LIN {X 0,Y 656.693,Z 410.418,A -85,B 0,C 180,E1 30799.109,E2 30799.109} C_VEL
LIN {X 0,Y 656.695,Z 410.425,A -85,B 0,C 180,E1 30796.088,E2 30796.088} C_VEL
LIN {X 0,Y 656.69,Z 410.427,A -85,B 0,C 180,E1 30793.023,E2 30793.023} C_VEL
LIN {X 0,Y 656.7,Z 410.423,A -85,B 0,C 180,E1 30789.996,E2 30789.996} C_VEL
LIN {X 0,Y 656.683,Z 410.43,A -85,B 0,C 180,E1 30786.896,E2 30786.896} C_VEL
LIN {X 0,Y 656.702,Z 410.42,A -85,B 0,C 180,E1 30783.841,E2 30783.841} C_VEL
LIN {X 0,Y 656.676,Z 410.43,A -85,B 0,C 180,E1 30780.785,E2 30780.785} C_VEL
LIN {X 0,Y 656.705,Z 410.416,A -85,B 0,C 180,E1 30777.819,E2 30777.819} C_VEL
LIN {X 0,Y 656.671,Z 410.43,A -85,B 0,C 180,E1 30774.758,E2 30774.758} C_VEL
LIN {X 0,Y 656.707,Z 410.411,A -85,B 0,C 180,E1 30771.763,E2 30771.763} C_VEL
LIN {X 0,Y 656.665,Z 410.429,A -85,B 0,C 180,E1 30768.672,E2 30768.672} C_VEL
LIN {X 0,Y 656.702,Z 410.411,A -85,B 0,C 180,E1 30765.72,E2 30765.72} C_VEL
LIN {X 0,Y 656.661,Z 410.426,A -85,B 0,C 180,E1 30762.636,E2 30762.636} C_VEL
LIN {X 0,Y 656.679,Z 410.421,A -85,B 0,C 180,E1 30759.779,E2 30759.779} C_VEL
LIN {X 0,Y 656.66,Z 410.417,A -85,B 0,C 180,E1 30756.663,E2 30756.663} C_VEL
LIN {X 0,Y 656.653,Z 410.429,A -85,B 0,C 180,E1 30753.892,E2 30753.892} C_VEL
LIN {X 0,Y 656.668,Z 410.427,A -85,B 0,C 180,E1 30750.74,E2 30750.74} C_VEL
LIN {X 0,Y 656.635,Z 410.428,A -85,B 0,C 180,E1 30748,E2 30748} C_VEL
LIN {X 0,Y 656.698,Z 410.433,A -85,B 0,C 180,E1 30744.969,E2 30744.969} C_VEL
LIN {X 0,Y 656.625,Z 410.434,A -85,B 0,C 180,E1 30742.074,E2 30742.074} C_VEL
LIN {X 0,Y 656.649,Z 410.429,A -85,B 0,C 180,E1 30740.539,E2 30740.539} C_VEL
LIN {X 0,Y 655.6,Z 410.557,A -85,B 0,C 180,E1 30739.867,E2 30739.867} C_VEL
LIN {X 0,Y 649.187,Z 411.313,A -85,B 0,C 180,E1 30737.983,E2 30737.983} C_VEL
LIN {X 0,Y 648.697,Z 411.374,A -85,B 0,C 180,E1 30737.493,E2 30737.493} C_VEL
LIN {X 0,Y 648.686,Z 411.423,A -85,B 0,C 180,E1 30734.288,E2 30734.288} C_VEL
LIN {X 0,Y 648.673,Z 411.379,A -85,B 0,C 180,E1 30731.617,E2 30731.617} C_VEL
LIN {X 0,Y 648.721,Z 411.408,A -85,B 0,C 180,E1 30728.606,E2 30728.606} C_VEL
LIN {X 0,Y 648.773,Z 411.633,A -85,B 0,C 180,E1 30726.726,E2 30726.726} C_VEL
LIN {X 0,Y 650.211,Z 415.779,A -85,B 0,C 180,E1 30726.237,E2 30726.237} C_VEL
LIN {X 0,Y 662.995,Z 436.741,A -85,B 0,C 180,E1 30725.041,E2 30725.041} C_VEL
LIN {X 0,Y 667.932,Z 445.525,A -85,B 0,C 180,E1 30724.59,E2 30724.59} C_VEL
LIN {X 0,Y 664.816,Z 693.939,A -85,B 0,C 180,E1 30721.53,E2 30721.53} C_VEL
LIN {X 0,Y 663.436,Z 804.05,A -85,B 0,C 180,E1 30720.173,E2 30720.173} C_VEL
LIN {X 0,Y 662.695,Z 829.21,A -85,B 0,C 180,E1 30719.71,E2 30719.71} C_VEL
LIN {X 0,Y 661.876,Z 849.807,A -85,B 0,C 180,E1 30719.2,E2 30719.2} C_VEL
LIN {X 0,Y 660.879,Z 872.181,A -85,B 0,C 180,E1 30718.512,E2 30718.512} C_VEL
LIN {X 0,Y 659.671,Z 893.971,A -85,B 0,C 180,E1 30717.683,E2 30717.683} C_VEL
LIN {X 0,Y 658.517,Z 914.637,A -85,B 0,C 180,E1 30716.757,E2 30716.757} C_VEL
LIN {X 0,Y 657.055,Z 937.416,A -85,B 0,C 180,E1 30715.553,E2 30715.553} C_VEL
LIN {X 0,Y 655.807,Z 956.221,A -85,B 0,C 180,E1 30714.405,E2 30714.405} C_VEL
LIN {X 0,Y 654.415,Z 977.19,A -85,B 0,C 180,E1 30712.931,E2 30712.931} C_VEL
LIN {X 0,Y 653.234,Z 994.357,A -85,B 0,C 180,E1 30711.553,E2 30711.553} C_VEL
LIN {X 0,Y 652.004,Z 1013.415,A -85,B 0,C 180,E1 30709.811,E2 30709.811} C_VEL
LIN {X 0,Y 651.067,Z 1028.308,A -85,B 0,C 180,E1 30708.258,E2 30708.258} C_VEL
LIN {X 0,Y 650.158,Z 1044.481,A -85,B 0,C 180,E1 30706.346,E2 30706.346} C_VEL
LIN {X 0,Y 649.48,Z 1057.15,A -85,B 0,C 180,E1 30704.625,E2 30704.625} C_VEL
LIN {X 0,Y 648.926,Z 1069.98,A -85,B 0,C 180,E1 30702.639,E2 30702.639} C_VEL
LIN {X 0,Y 648.524,Z 1080.788,A -85,B 0,C 180,E1 30700.662,E2 30700.662} C_VEL
LIN {X 0,Y 648.247,Z 1090.431,A -85,B 0,C 180,E1 30698.605,E2 30698.605} C_VEL
LIN {X 0,Y 648.052,Z 1098.176,A -85,B 0,C 180,E1 30696.556,E2 30696.556} C_VEL
LIN {X 0,Y 647.96,Z 1103.94,A -85,B 0,C 180,E1 30694.691,E2 30694.691} C_VEL
LIN {X 0,Y 647.925,Z 1109.279,A -85,B 0,C 180,E1 30692.388,E2 30692.388} C_VEL
LIN {X 0,Y 647.914,Z 1112.302,A -85,B 0,C 180,E1 30690.442,E2 30690.442} C_VEL
LIN {X 0,Y 647.894,Z 1114.159,A -85,B 0,C 180,E1 30688.32,E2 30688.32} C_VEL
LIN {X 0,Y 647.892,Z 1114.337,A -85,B 0,C 180,E1 30686.284,E2 30686.284} C_VEL
LIN {X 0,Y 647.905,Z 1113.249,A -85,B 0,C 180,E1 30684.332,E2 30684.332} C_VEL
LIN {X 0,Y 647.924,Z 1110.328,A -85,B 0,C 180,E1 30682.106,E2 30682.106} C_VEL
LIN {X 0,Y 647.93,Z 1106.499,A -85,B 0,C 180,E1 30680.227,E2 30680.227} C_VEL
LIN {X 0,Y 647.996,Z 1100.901,A -85,B 0,C 180,E1 30678.157,E2 30678.157} C_VEL
LIN {X 0,Y 648.149,Z 1093.476,A -85,B 0,C 180,E1 30676.074,E2 30676.074} C_VEL
LIN {X 0,Y 648.371,Z 1085.278,A -85,B 0,C 180,E1 30674.159,E2 30674.159} C_VEL
LIN {X 0,Y 648.734,Z 1074.384,A -85,B 0,C 180,E1 30672.046,E2 30672.046} C_VEL
LIN {X 0,Y 649.186,Z 1063.508,A -85,B 0,C 180,E1 30670.234,E2 30670.234} C_VEL
LIN {X 0,Y 649.864,Z 1049.605,A -85,B 0,C 180,E1 30668.235,E2 30668.235} C_VEL
LIN {X 0,Y 650.618,Z 1036.132,A -85,B 0,C 180,E1 30666.544,E2 30666.544} C_VEL
LIN {X 0,Y 651.643,Z 1018.935,A -85,B 0,C 180,E1 30664.653,E2 30664.653} C_VEL
LIN {X 0,Y 652.668,Z 1003.148,A -85,B 0,C 180,E1 30663.132,E2 30663.132} C_VEL
LIN {X 0,Y 653.958,Z 983.638,A -85,B 0,C 180,E1 30661.474,E2 30661.474} C_VEL
LIN {X 0,Y 655.214,Z 965.251,A -85,B 0,C 180,E1 30660.115,E2 30660.115} C_VEL
LIN {X 0,Y 656.661,Z 943.663,A -85,B 0,C 180,E1 30658.719,E2 30658.719} C_VEL
LIN {X 0,Y 657.924,Z 923.66,A -85,B 0,C 180,E1 30657.607,E2 30657.607} C_VEL
LIN {X 0,Y 659.328,Z 900.994,A -85,B 0,C 180,E1 30656.522,E2 30656.522} C_VEL
LIN {X 0,Y 660.467,Z 879.681,A -85,B 0,C 180,E1 30655.672,E2 30655.672} C_VEL
LIN {X 0,Y 661.604,Z 856.553,A -85,B 0,C 180,E1 30654.896,E2 30654.896} C_VEL
LIN {X 0,Y 662.536,Z 832.984,A -85,B 0,C 180,E1 30654.285,E2 30654.285} C_VEL
LIN {X 0,Y 663.294,Z 810.621,A -85,B 0,C 180,E1 30653.841,E2 30653.841} C_VEL
LIN {X 0,Y 663.84,Z 776.914,A -85,B 0,C 180,E1 30653.386,E2 30653.386} C_VEL
LIN {X 0,Y 666.852,Z 528.949,A -85,B 0,C 180,E1 30650.355,E2 30650.355} C_VEL
LIN {X 0,Y 667.836,Z 445.069,A -85,B 0,C 180,E1 30649.307,E2 30649.307} C_VEL
LIN {X 0,Y 654.643,Z 422.915,A -85,B 0,C 180,E1 30648.092,E2 30648.092} C_VEL
LIN {X 0,Y 650.084,Z 415.41,A -85,B 0,C 180,E1 30647.628,E2 30647.628} C_VEL
LIN {X 0,Y 648.768,Z 411.552,A -85,B 0,C 180,E1 30647.121,E2 30647.121} C_VEL
LIN {X 0,Y 648.675,Z 411.43,A -85,B 0,C 180,E1 30644.165,E2 30644.165} C_VEL
LIN {X 0,Y 648.698,Z 411.385,A -85,B 0,C 180,E1 30641.486,E2 30641.486} C_VEL
LIN {X 0,Y 648.696,Z 411.42,A -85,B 0,C 180,E1 30638.319,E2 30638.319} C_VEL
LIN {X 0,Y 648.687,Z 411.38,A -85,B 0,C 180,E1 30635.637,E2 30635.637} C_VEL
LIN {X 0,Y 648.737,Z 411.417,A -85,B 0,C 180,E1 30632.532,E2 30632.532} C_VEL
LIN {X 0,Y 648.69,Z 411.378,A -85,B 0,C 180,E1 30629.758,E2 30629.758} C_VEL
LIN {X 0,Y 648.773,Z 411.415,A -85,B 0,C 180,E1 30626.829,E2 30626.829} C_VEL
LIN {X 0,Y 648.704,Z 411.411,A -85,B 0,C 180,E1 30623.818,E2 30623.818} C_VEL
LIN {X 0,Y 648.746,Z 411.416,A -85,B 0,C 180,E1 30621.046,E2 30621.046} C_VEL
LIN {X 0,Y 648.723,Z 411.418,A -85,B 0,C 180,E1 30617.955,E2 30617.955} C_VEL
LIN {X 0,Y 648.738,Z 411.409,A -85,B 0,C 180,E1 30615.098,E2 30615.098} C_VEL
LIN {X 0,Y 648.733,Z 411.407,A -85,B 0,C 180,E1 30611.919,E2 30611.919} C_VEL
LIN {X 0,Y 648.753,Z 411.422,A -85,B 0,C 180,E1 30608.956,E2 30608.956} C_VEL
LIN {X 0,Y 648.735,Z 411.411,A -85,B 0,C 180,E1 30605.75,E2 30605.75} C_VEL
LIN {X 0,Y 648.763,Z 411.407,A -85,B 0,C 180,E1 30602.739,E2 30602.739} C_VEL
LIN {X 0,Y 648.741,Z 411.414,A -85,B 0,C 180,E1 30599.647,E2 30599.647} C_VEL
LIN {X 0,Y 648.765,Z 411.407,A -85,B 0,C 180,E1 30596.554,E2 30596.554} C_VEL
LIN {X 0,Y 648.742,Z 411.411,A -85,B 0,C 180,E1 30593.451,E2 30593.451} C_VEL
LIN {X 0,Y 648.763,Z 411.419,A -85,B 0,C 180,E1 30590.418,E2 30590.418} C_VEL
LIN {X 0,Y 648.747,Z 411.402,A -85,B 0,C 180,E1 30587.324,E2 30587.324} C_VEL
LIN {X 0,Y 648.757,Z 411.411,A -85,B 0,C 180,E1 30584.353,E2 30584.353} C_VEL
LIN {X 0,Y 648.754,Z 411.415,A -85,B 0,C 180,E1 30581.209,E2 30581.209} C_VEL
LIN {X 0,Y 648.749,Z 411.401,A -85,B 0,C 180,E1 30578.195,E2 30578.195} C_VEL
LIN {X 0,Y 648.759,Z 411.416,A -85,B 0,C 180,E1 30575.117,E2 30575.117} C_VEL
LIN {X 0,Y 648.745,Z 411.417,A -85,B 0,C 180,E1 30572.025,E2 30572.025} C_VEL
LIN {X 0,Y 648.762,Z 411.405,A -85,B 0,C 180,E1 30568.973,E2 30568.973} C_VEL
LIN {X 0,Y 648.738,Z 411.417,A -85,B 0,C 180,E1 30565.98,E2 30565.98} C_VEL
LIN {X 0,Y 648.768,Z 411.415,A -85,B 0,C 180,E1 30562.942,E2 30562.942} C_VEL
LIN {X 0,Y 648.732,Z 411.418,A -85,B 0,C 180,E1 30559.889,E2 30559.889} C_VEL
LIN {X 0,Y 648.768,Z 411.405,A -85,B 0,C 180,E1 30556.932,E2 30556.932} C_VEL
LIN {X 0,Y 648.725,Z 411.416,A -85,B 0,C 180,E1 30553.835,E2 30553.835} C_VEL
LIN {X 0,Y 648.802,Z 411.636,A -85,B 0,C 180,E1 30552.719,E2 30552.719} C_VEL
LIN {X 0,Y 656.404,Z 431.204,A -85,B 0,C 180,E1 30550.46,E2 30550.46} C_VEL
LIN {X 0,Y 661.805,Z 445.758,A -85,B 0,C 180,E1 30548.914,E2 30548.914} C_VEL
LIN {X 0,Y 661.676,Z 451.804,A -85,B 0,C 180,E1 30548.484,E2 30548.484} C_VEL
LIN {X 0,Y 667.819,Z 478.941,A -85,B 0,C 180,E1 30547.699,E2 30547.699} C_VEL
LIN {X 0,Y 664.86,Z 722.844,A -85,B 0,C 180,E1 30544.702,E2 30544.702} C_VEL
LIN {X 0,Y 663.414,Z 843.427,A -85,B 0,C 180,E1 30543.221,E2 30543.221} C_VEL
LIN {X 0,Y 662.661,Z 868.958,A -85,B 0,C 180,E1 30542.754,E2 30542.754} C_VEL
LIN {X 0,Y 661.847,Z 889.812,A -85,B 0,C 180,E1 30542.241,E2 30542.241} C_VEL
LIN {X 0,Y 660.852,Z 912.607,A -85,B 0,C 180,E1 30541.543,E2 30541.543} C_VEL
LIN {X 0,Y 659.662,Z 934.199,A -85,B 0,C 180,E1 30540.718,E2 30540.718} C_VEL
LIN {X 0,Y 658.536,Z 954.262,A -85,B 0,C 180,E1 30539.819,E2 30539.819} C_VEL
LIN {X 0,Y 657.113,Z 976.679,A -85,B 0,C 180,E1 30538.641,E2 30538.641} C_VEL
LIN {X 0,Y 655.816,Z 996.099,A -85,B 0,C 180,E1 30537.458,E2 30537.458} C_VEL
LIN {X 0,Y 654.402,Z 1017.39,A -85,B 0,C 180,E1 30535.961,E2 30535.961} C_VEL
LIN {X 0,Y 653.209,Z 1034.842,A -85,B 0,C 180,E1 30534.557,E2 30534.557} C_VEL
LIN {X 0,Y 651.983,Z 1053.748,A -85,B 0,C 180,E1 30532.823,E2 30532.823} C_VEL
LIN {X 0,Y 651.037,Z 1068.783,A -85,B 0,C 180,E1 30531.251,E2 30531.251} C_VEL
LIN {X 0,Y 650.117,Z 1085.113,A -85,B 0,C 180,E1 30529.31,E2 30529.31} C_VEL
LIN {X 0,Y 649.45,Z 1097.884,A -85,B 0,C 180,E1 30527.563,E2 30527.563} C_VEL
LIN {X 0,Y 648.86,Z 1111.247,A -85,B 0,C 180,E1 30525.462,E2 30525.462} C_VEL
LIN {X 0,Y 648.488,Z 1121.103,A -85,B 0,C 180,E1 30523.645,E2 30523.645} C_VEL
LIN {X 0,Y 648.218,Z 1130.768,A -85,B 0,C 180,E1 30521.568,E2 30521.568} C_VEL
LIN {X 0,Y 648.055,Z 1138.514,A -85,B 0,C 180,E1 30519.503,E2 30519.503} C_VEL
LIN {X 0,Y 647.941,Z 1144.761,A -85,B 0,C 180,E1 30517.448,E2 30517.448} C_VEL
LIN {X 0,Y 647.899,Z 1149.496,A -85,B 0,C 180,E1 30515.313,E2 30515.313} C_VEL
LIN {X 0,Y 647.909,Z 1152.35,A -85,B 0,C 180,E1 30513.451,E2 30513.451} C_VEL
LIN {X 0,Y 647.909,Z 1154.192,A -85,B 0,C 180,E1 30511.238,E2 30511.238} C_VEL
LIN {X 0,Y 647.885,Z 1154.328,A -85,B 0,C 180,E1 30509.293,E2 30509.293} C_VEL
LIN {X 0,Y 647.888,Z 1153.225,A -85,B 0,C 180,E1 30507.346,E2 30507.346} C_VEL
LIN {X 0,Y 647.903,Z 1150.292,A -85,B 0,C 180,E1 30505.131,E2 30505.131} C_VEL
LIN {X 0,Y 647.939,Z 1146.689,A -85,B 0,C 180,E1 30503.354,E2 30503.354} C_VEL
LIN {X 0,Y 648,Z 1140.935,A -85,B 0,C 180,E1 30501.213,E2 30501.213} C_VEL
LIN {X 0,Y 648.142,Z 1133.603,A -85,B 0,C 180,E1 30499.152,E2 30499.152} C_VEL
LIN {X 0,Y 648.372,Z 1125.529,A -85,B 0,C 180,E1 30497.26,E2 30497.26} C_VEL
LIN {X 0,Y 648.748,Z 1114.436,A -85,B 0,C 180,E1 30495.1,E2 30495.1} C_VEL
LIN {X 0,Y 649.198,Z 1103.393,A -85,B 0,C 180,E1 30493.261,E2 30493.261} C_VEL
LIN {X 0,Y 649.877,Z 1089.323,A -85,B 0,C 180,E1 30491.242,E2 30491.242} C_VEL
LIN {X 0,Y 650.67,Z 1075.307,A -85,B 0,C 180,E1 30489.49,E2 30489.49} C_VEL
LIN {X 0,Y 651.686,Z 1058.305,A -85,B 0,C 180,E1 30487.635,E2 30487.635} C_VEL
LIN {X 0,Y 652.726,Z 1042.29,A -85,B 0,C 180,E1 30486.098,E2 30486.098} C_VEL
LIN {X 0,Y 654.04,Z 1022.359,A -85,B 0,C 180,E1 30484.421,E2 30484.421} C_VEL
LIN {X 0,Y 655.275,Z 1004.392,A -85,B 0,C 180,E1 30483.1,E2 30483.1} C_VEL
LIN {X 0,Y 656.73,Z 982.354,A -85,B 0,C 180,E1 30481.688,E2 30481.688} C_VEL
LIN {X 0,Y 657.988,Z 962.741,A -85,B 0,C 180,E1 30480.604,E2 30480.604} C_VEL
LIN {X 0,Y 659.437,Z 938.724,A -85,B 0,C 180,E1 30479.472,E2 30479.472} C_VEL
LIN {X 0,Y 660.468,Z 919.672,A -85,B 0,C 180,E1 30478.716,E2 30478.716} C_VEL
LIN {X 0,Y 661.556,Z 897.1,A -85,B 0,C 180,E1 30477.96,E2 30477.96} C_VEL
LIN {X 0,Y 662.486,Z 873.196,A -85,B 0,C 180,E1 30477.34,E2 30477.34} C_VEL
LIN {X 0,Y 663.235,Z 851.125,A -85,B 0,C 180,E1 30476.901,E2 30476.901} C_VEL
LIN {X 0,Y 663.789,Z 818.284,A -85,B 0,C 180,E1 30476.453,E2 30476.453} C_VEL
LIN {X 0,Y 666.423,Z 587.514,A -85,B 0,C 180,E1 30473.641,E2 30473.641} C_VEL
LIN {X 0,Y 667.672,Z 477.41,A -85,B 0,C 180,E1 30472.271,E2 30472.271} C_VEL
LIN {X 0,Y 661.622,Z 451.279,A -85,B 0,C 180,E1 30471.49,E2 30471.49} C_VEL
LIN {X 0,Y 661.73,Z 445.472,A -85,B 0,C 180,E1 30471.054,E2 30471.054} C_VEL
LIN {X 0,Y 652.71,Z 421.722,A -85,B 0,C 180,E1 30468.513,E2 30468.513} C_VEL
LIN {X 0,Y 648.798,Z 411.615,A -85,B 0,C 180,E1 30467.35,E2 30467.35} C_VEL
LIN {X 0,Y 648.726,Z 411.423,A -85,B 0,C 180,E1 30464.343,E2 30464.343} C_VEL
LIN {X 0,Y 648.764,Z 411.366,A -85,B 0,C 180,E1 30461.359,E2 30461.359} C_VEL
LIN {X 0,Y 648.733,Z 411.42,A -85,B 0,C 180,E1 30458.287,E2 30458.287} C_VEL
LIN {X 0,Y 648.766,Z 411.421,A -85,B 0,C 180,E1 30455.307,E2 30455.307} C_VEL
LIN {X 0,Y 648.738,Z 411.409,A -85,B 0,C 180,E1 30452.202,E2 30452.202} C_VEL
LIN {X 0,Y 648.761,Z 411.404,A -85,B 0,C 180,E1 30449.247,E2 30449.247} C_VEL
LIN {X 0,Y 648.748,Z 411.417,A -85,B 0,C 180,E1 30446.155,E2 30446.155} C_VEL
LIN {X 0,Y 648.759,Z 411.411,A -85,B 0,C 180,E1 30443.142,E2 30443.142} C_VEL
LIN {X 0,Y 648.752,Z 411.412,A -85,B 0,C 180,E1 30440.103,E2 30440.103} C_VEL
LIN {X 0,Y 648.754,Z 411.419,A -85,B 0,C 180,E1 30437.028,E2 30437.028} C_VEL
LIN {X 0,Y 648.754,Z 411.401,A -85,B 0,C 180,E1 30434.003,E2 30434.003} C_VEL
LIN {X 0,Y 648.748,Z 411.416,A -85,B 0,C 180,E1 30430.928,E2 30430.928} C_VEL
LIN {X 0,Y 648.76,Z 411.401,A -85,B 0,C 180,E1 30427.884,E2 30427.884} C_VEL
LIN {X 0,Y 648.742,Z 411.413,A -85,B 0,C 180,E1 30424.863,E2 30424.863} C_VEL
LIN {X 0,Y 648.763,Z 411.406,A -85,B 0,C 180,E1 30421.766,E2 30421.766} C_VEL
LIN {X 0,Y 648.735,Z 411.409,A -85,B 0,C 180,E1 30418.764,E2 30418.764} C_VEL
LIN {X 0,Y 648.767,Z 411.409,A -85,B 0,C 180,E1 30415.69,E2 30415.69} C_VEL
LIN {X 0,Y 648.727,Z 411.405,A -85,B 0,C 180,E1 30412.65,E2 30412.65} C_VEL
LIN {X 0,Y 648.771,Z 411.412,A -85,B 0,C 180,E1 30409.611,E2 30409.611} C_VEL
LIN {X 0,Y 648.719,Z 411.404,A -85,B 0,C 180,E1 30406.541,E2 30406.541} C_VEL
LIN {X 0,Y 648.768,Z 411.415,A -85,B 0,C 180,E1 30403.618,E2 30403.618} C_VEL
LIN {X 0,Y 648.718,Z 411.413,A -85,B 0,C 180,E1 30400.553,E2 30400.553} C_VEL
LIN {X 0,Y 648.752,Z 411.415,A -85,B 0,C 180,E1 30397.632,E2 30397.632} C_VEL
LIN {X 0,Y 648.712,Z 411.421,A -85,B 0,C 180,E1 30394.53,E2 30394.53} C_VEL
LIN {X 0,Y 648.72,Z 411.411,A -85,B 0,C 180,E1 30391.758,E2 30391.758} C_VEL
LIN {X 0,Y 648.716,Z 411.419,A -85,B 0,C 180,E1 30388.602,E2 30388.602} C_VEL
LIN {X 0,Y 648.698,Z 411.419,A -85,B 0,C 180,E1 30385.866,E2 30385.866} C_VEL
LIN {X 0,Y 648.746,Z 411.412,A -85,B 0,C 180,E1 30382.829,E2 30382.829} C_VEL
LIN {X 0,Y 648.683,Z 411.417,A -85,B 0,C 180,E1 30380.116,E2 30380.116} C_VEL
LIN {X 0,Y 648.697,Z 411.374,A -85,B 0,C 180,E1 30377.493,E2 30377.493} C_VEL
LIN {X 0,Y 647.763,Z 411.505,A -85,B 0,C 180,E1 30376.812,E2 30376.812} C_VEL
LIN {X 0,Y 641.232,Z 412.36,A -85,B 0,C 180,E1 30374.856,E2 30374.856} C_VEL
LIN {X 0,Y 640.759,Z 412.412,A -85,B 0,C 180,E1 30374.409,E2 30374.409} C_VEL
LIN {X 0,Y 640.731,Z 412.365,A -85,B 0,C 180,E1 30371.667,E2 30371.667} C_VEL
LIN {X 0,Y 640.784,Z 412.396,A -85,B 0,C 180,E1 30368.621,E2 30368.621} C_VEL
LIN {X 0,Y 640.782,Z 412.588,A -85,B 0,C 180,E1 30367.261,E2 30367.261} C_VEL
LIN {X 0,Y 642.1,Z 415.927,A -85,B 0,C 180,E1 30366.83,E2 30366.83} C_VEL
LIN {X 0,Y 657.916,Z 442.03,A -85,B 0,C 180,E1 30365.32,E2 30365.32} C_VEL
LIN {X 0,Y 661.574,Z 448.558,A -85,B 0,C 180,E1 30364.979,E2 30364.979} C_VEL
LIN {X 0,Y 658.205,Z 697.351,A -85,B 0,C 180,E1 30361.887,E2 30361.887} C_VEL
LIN {X 0,Y 656.752,Z 804.435,A -85,B 0,C 180,E1 30360.554,E2 30360.554} C_VEL
LIN {X 0,Y 655.966,Z 829.558,A -85,B 0,C 180,E1 30360.087,E2 30360.087} C_VEL
LIN {X 0,Y 655.103,Z 850.036,A -85,B 0,C 180,E1 30359.576,E2 30359.576} C_VEL
LIN {X 0,Y 653.994,Z 872.934,A -85,B 0,C 180,E1 30358.863,E2 30358.863} C_VEL
LIN {X 0,Y 652.654,Z 895.029,A -85,B 0,C 180,E1 30358.007,E2 30358.007} C_VEL
LIN {X 0,Y 651.292,Z 917.442,A -85,B 0,C 180,E1 30356.979,E2 30356.979} C_VEL
LIN {X 0,Y 649.77,Z 938.894,A -85,B 0,C 180,E1 30355.812,E2 30355.812} C_VEL
LIN {X 0,Y 648.364,Z 958.816,A -85,B 0,C 180,E1 30354.571,E2 30354.571} C_VEL
LIN {X 0,Y 646.886,Z 978.905,A -85,B 0,C 180,E1 30353.117,E2 30353.117} C_VEL
LIN {X 0,Y 645.557,Z 997.014,A -85,B 0,C 180,E1 30351.632,E2 30351.632} C_VEL
LIN {X 0,Y 644.302,Z 1014.725,A -85,B 0,C 180,E1 30349.963,E2 30349.963} C_VEL
LIN {X 0,Y 643.303,Z 1029.505,A -85,B 0,C 180,E1 30348.393,E2 30348.393} C_VEL
LIN {X 0,Y 642.32,Z 1045.482,A -85,B 0,C 180,E1 30346.458,E2 30346.458} C_VEL
LIN {X 0,Y 641.595,Z 1058.05,A -85,B 0,C 180,E1 30344.716,E2 30344.716} C_VEL
LIN {X 0,Y 640.969,Z 1071.232,A -85,B 0,C 180,E1 30342.615,E2 30342.615} C_VEL
LIN {X 0,Y 640.565,Z 1081.438,A -85,B 0,C 180,E1 30340.705,E2 30340.705} C_VEL
LIN {X 0,Y 640.25,Z 1091.297,A -85,B 0,C 180,E1 30338.532,E2 30338.532} C_VEL
LIN {X 0,Y 640.061,Z 1098.607,A -85,B 0,C 180,E1 30336.548,E2 30336.548} C_VEL
LIN {X 0,Y 639.962,Z 1104.807,A -85,B 0,C 180,E1 30334.481,E2 30334.481} C_VEL
LIN {X 0,Y 639.925,Z 1109.505,A -85,B 0,C 180,E1 30332.328,E2 30332.328} C_VEL
LIN {X 0,Y 639.914,Z 1112.35,A -85,B 0,C 180,E1 30330.448,E2 30330.448} C_VEL
LIN {X 0,Y 639.903,Z 1114.192,A -85,B 0,C 180,E1 30328.209,E2 30328.209} C_VEL
LIN {X 0,Y 639.893,Z 1114.327,A -85,B 0,C 180,E1 30326.237,E2 30326.237} C_VEL
LIN {X 0,Y 639.906,Z 1113.151,A -85,B 0,C 180,E1 30324.171,E2 30324.171} C_VEL
LIN {X 0,Y 639.925,Z 1110.26,A -85,B 0,C 180,E1 30322.006,E2 30322.006} C_VEL
LIN {X 0,Y 639.943,Z 1106.409,A -85,B 0,C 180,E1 30320.103,E2 30320.103} C_VEL
LIN {X 0,Y 640.018,Z 1100.466,A -85,B 0,C 180,E1 30317.916,E2 30317.916} C_VEL
LIN {X 0,Y 640.177,Z 1093.322,A -85,B 0,C 180,E1 30315.898,E2 30315.898} C_VEL
LIN {X 0,Y 640.435,Z 1085.1,A -85,B 0,C 180,E1 30313.958,E2 30313.958} C_VEL
LIN {X 0,Y 640.838,Z 1074.156,A -85,B 0,C 180,E1 30311.817,E2 30311.817} C_VEL
LIN {X 0,Y 641.35,Z 1062.996,A -85,B 0,C 180,E1 30309.941,E2 30309.941} C_VEL
LIN {X 0,Y 642.096,Z 1048.896,A -85,B 0,C 180,E1 30307.904,E2 30307.904} C_VEL
LIN {X 0,Y 642.97,Z 1034.999,A -85,B 0,C 180,E1 30306.151,E2 30306.151} C_VEL
LIN {X 0,Y 644.073,Z 1018.047,A -85,B 0,C 180,E1 30304.284,E2 30304.284} C_VEL
LIN {X 0,Y 645.158,Z 1002.693,A -85,B 0,C 180,E1 30302.793,E2 30302.793} C_VEL
LIN {X 0,Y 646.606,Z 982.537,A -85,B 0,C 180,E1 30301.074,E2 30301.074} C_VEL
LIN {X 0,Y 647.879,Z 965.334,A -85,B 0,C 180,E1 30299.793,E2 30299.793} C_VEL
LIN {X 0,Y 649.386,Z 944.599,A -85,B 0,C 180,E1 30298.432,E2 30298.432} C_VEL
LIN {X 0,Y 650.726,Z 924.95,A -85,B 0,C 180,E1 30297.323,E2 30297.323} C_VEL
LIN {X 0,Y 652.231,Z 902.871,A -85,B 0,C 180,E1 30296.239,E2 30296.239} C_VEL
LIN {X 0,Y 653.533,Z 880.731,A -85,B 0,C 180,E1 30295.335,E2 30295.335} C_VEL
LIN {X 0,Y 654.636,Z 860.09,A -85,B 0,C 180,E1 30294.628,E2 30294.628} C_VEL
LIN {X 0,Y 655.729,Z 835.009,A -85,B 0,C 180,E1 30293.946,E2 30293.946} C_VEL
LIN {X 0,Y 656.506,Z 813.457,A -85,B 0,C 180,E1 30293.505,E2 30293.505} C_VEL
LIN {X 0,Y 657.125,Z 782.42,A -85,B 0,C 180,E1 30293.064,E2 30293.064} C_VEL
LIN {X 0,Y 660.384,Z 533.527,A -85,B 0,C 180,E1 30289.994,E2 30289.994} C_VEL
LIN {X 0,Y 661.464,Z 448.008,A -85,B 0,C 180,E1 30288.916,E2 30288.916} C_VEL
LIN {X 0,Y 647.578,Z 424.844,A -85,B 0,C 180,E1 30287.599,E2 30287.599} C_VEL
LIN {X 0,Y 642.127,Z 415.951,A -85,B 0,C 180,E1 30287.043,E2 30287.043} C_VEL
LIN {X 0,Y 640.778,Z 412.568,A -85,B 0,C 180,E1 30286.58,E2 30286.58} C_VEL
LIN {X 0,Y 640.739,Z 412.419,A -85,B 0,C 180,E1 30283.858,E2 30283.858} C_VEL
LIN {X 0,Y 640.805,Z 412.374,A -85,B 0,C 180,E1 30280.819,E2 30280.819} C_VEL
LIN {X 0,Y 640.744,Z 412.408,A -85,B 0,C 180,E1 30277.995,E2 30277.995} C_VEL
LIN {X 0,Y 640.796,Z 412.37,A -85,B 0,C 180,E1 30275.15,E2 30275.15} C_VEL
LIN {X 0,Y 640.759,Z 412.407,A -85,B 0,C 180,E1 30272.076,E2 30272.076} C_VEL
LIN {X 0,Y 640.773,Z 412.362,A -85,B 0,C 180,E1 30269.339,E2 30269.339} C_VEL
LIN {X 0,Y 640.775,Z 412.41,A -85,B 0,C 180,E1 30266.107,E2 30266.107} C_VEL
LIN {X 0,Y 640.777,Z 412.401,A -85,B 0,C 180,E1 30263.35,E2 30263.35} C_VEL
LIN {X 0,Y 640.795,Z 412.395,A -85,B 0,C 180,E1 30260.173,E2 30260.173} C_VEL
LIN {X 0,Y 640.788,Z 412.411,A -85,B 0,C 180,E1 30257.259,E2 30257.259} C_VEL
LIN {X 0,Y 640.797,Z 412.406,A -85,B 0,C 180,E1 30253.996,E2 30253.996} C_VEL
LIN {X 0,Y 640.803,Z 412.396,A -85,B 0,C 180,E1 30251.045,E2 30251.045} C_VEL
LIN {X 0,Y 640.801,Z 412.4,A -85,B 0,C 180,E1 30247.892,E2 30247.892} C_VEL
LIN {X 0,Y 640.821,Z 412.407,A -85,B 0,C 180,E1 30244.833,E2 30244.833} C_VEL
LIN {X 0,Y 640.801,Z 412.389,A -85,B 0,C 180,E1 30241.699,E2 30241.699} C_VEL
LIN {X 0,Y 640.828,Z 412.4,A -85,B 0,C 180,E1 30238.659,E2 30238.659} C_VEL
LIN {X 0,Y 640.805,Z 412.4,A -85,B 0,C 180,E1 30235.525,E2 30235.525} C_VEL
LIN {X 0,Y 640.824,Z 412.393,A -85,B 0,C 180,E1 30232.469,E2 30232.469} C_VEL
LIN {X 0,Y 640.808,Z 412.404,A -85,B 0,C 180,E1 30229.39,E2 30229.39} C_VEL
LIN {X 0,Y 640.818,Z 412.408,A -85,B 0,C 180,E1 30226.28,E2 30226.28} C_VEL
LIN {X 0,Y 640.81,Z 412.394,A -85,B 0,C 180,E1 30223.222,E2 30223.222} C_VEL
LIN {X 0,Y 640.813,Z 412.402,A -85,B 0,C 180,E1 30220.202,E2 30220.202} C_VEL
LIN {X 0,Y 640.817,Z 412.393,A -85,B 0,C 180,E1 30217.137,E2 30217.137} C_VEL
LIN {X 0,Y 640.807,Z 412.392,A -85,B 0,C 180,E1 30214.094,E2 30214.094} C_VEL
LIN {X 0,Y 640.823,Z 412.404,A -85,B 0,C 180,E1 30211.073,E2 30211.073} C_VEL
LIN {X 0,Y 640.802,Z 412.397,A -85,B 0,C 180,E1 30208.064,E2 30208.064} C_VEL
LIN {X 0,Y 640.826,Z 412.396,A -85,B 0,C 180,E1 30205.002,E2 30205.002} C_VEL
LIN {X 0,Y 640.796,Z 412.404,A -85,B 0,C 180,E1 30201.949,E2 30201.949} C_VEL
LIN {X 0,Y 640.832,Z 412.408,A -85,B 0,C 180,E1 30198.906,E2 30198.906} C_VEL
LIN {X 0,Y 640.791,Z 412.411,A -85,B 0,C 180,E1 30195.872,E2 30195.872} C_VEL
LIN {X 0,Y 640.832,Z 412.643,A -85,B 0,C 180,E1 30193.278,E2 30193.278} C_VEL
LIN {X 0,Y 648.267,Z 431.418,A -85,B 0,C 180,E1 30191.041,E2 30191.041} C_VEL
LIN {X 0,Y 654.807,Z 449.36,A -85,B 0,C 180,E1 30189.098,E2 30189.098} C_VEL
LIN {X 0,Y 654.941,Z 452,A -85,B 0,C 180,E1 30188.944,E2 30188.944} C_VEL
LIN {X 0,Y 661.443,Z 480.54,A -85,B 0,C 180,E1 30188.101,E2 30188.101} C_VEL
LIN {X 0,Y 658.254,Z 723.423,A -85,B 0,C 180,E1 30185.089,E2 30185.089} C_VEL
LIN {X 0,Y 656.694,Z 843.157,A -85,B 0,C 180,E1 30183.605,E2 30183.605} C_VEL
LIN {X 0,Y 655.883,Z 868.783,A -85,B 0,C 180,E1 30183.133,E2 30183.133} C_VEL
LIN {X 0,Y 655.024,Z 889.289,A -85,B 0,C 180,E1 30182.625,E2 30182.625} C_VEL
LIN {X 0,Y 653.943,Z 912.355,A -85,B 0,C 180,E1 30181.915,E2 30181.915} C_VEL
LIN {X 0,Y 652.604,Z 935.229,A -85,B 0,C 180,E1 30181.036,E2 30181.036} C_VEL
LIN {X 0,Y 651.358,Z 956.268,A -85,B 0,C 180,E1 30180.08,E2 30180.08} C_VEL
LIN {X 0,Y 649.815,Z 978.321,A -85,B 0,C 180,E1 30178.891,E2 30178.891} C_VEL
LIN {X 0,Y 648.445,Z 997.452,A -85,B 0,C 180,E1 30177.704,E2 30177.704} C_VEL
LIN {X 0,Y 646.955,Z 1017.996,A -85,B 0,C 180,E1 30176.233,E2 30176.233} C_VEL
LIN {X 0,Y 645.705,Z 1035.015,A -85,B 0,C 180,E1 30174.846,E2 30174.846} C_VEL
LIN {X 0,Y 644.313,Z 1054.6,A -85,B 0,C 180,E1 30173.021,E2 30173.021} C_VEL
LIN {X 0,Y 643.279,Z 1069.863,A -85,B 0,C 180,E1 30171.398,E2 30171.398} C_VEL
LIN {X 0,Y 642.297,Z 1085.818,A -85,B 0,C 180,E1 30169.46,E2 30169.46} C_VEL
LIN {X 0,Y 641.574,Z 1098.517,A -85,B 0,C 180,E1 30167.692,E2 30167.692} C_VEL
LIN {X 0,Y 640.936,Z 1111.768,A -85,B 0,C 180,E1 30165.565,E2 30165.565} C_VEL
LIN {X 0,Y 640.536,Z 1121.561,A -85,B 0,C 180,E1 30163.726,E2 30163.726} C_VEL
LIN {X 0,Y 640.242,Z 1131.124,A -85,B 0,C 180,E1 30161.623,E2 30161.623} C_VEL
LIN {X 0,Y 640.066,Z 1138.513,A -85,B 0,C 180,E1 30159.622,E2 30159.622} C_VEL
LIN {X 0,Y 639.947,Z 1144.507,A -85,B 0,C 180,E1 30157.632,E2 30157.632} C_VEL
LIN {X 0,Y 639.905,Z 1149.336,A -85,B 0,C 180,E1 30155.47,E2 30155.47} C_VEL
LIN {X 0,Y 639.913,Z 1152.238,A -85,B 0,C 180,E1 30153.583,E2 30153.583} C_VEL
LIN {X 0,Y 639.904,Z 1154.169,A -85,B 0,C 180,E1 30151.343,E2 30151.343} C_VEL
LIN {X 0,Y 639.883,Z 1154.35,A -85,B 0,C 180,E1 30149.373,E2 30149.373} C_VEL
LIN {X 0,Y 639.897,Z 1153.361,A -85,B 0,C 180,E1 30147.492,E2 30147.492} C_VEL
LIN {X 0,Y 639.912,Z 1150.609,A -85,B 0,C 180,E1 30145.25,E2 30145.25} C_VEL
LIN {X 0,Y 639.941,Z 1146.896,A -85,B 0,C 180,E1 30143.36,E2 30143.36} C_VEL
LIN {X 0,Y 640.002,Z 1141.71,A -85,B 0,C 180,E1 30141.374,E2 30141.374} C_VEL
LIN {X 0,Y 640.156,Z 1134.309,A -85,B 0,C 180,E1 30139.197,E2 30139.197} C_VEL
LIN {X 0,Y 640.392,Z 1126.346,A -85,B 0,C 180,E1 30137.282,E2 30137.282} C_VEL
LIN {X 0,Y 640.799,Z 1115.378,A -85,B 0,C 180,E1 30135.08,E2 30135.08} C_VEL
LIN {X 0,Y 641.281,Z 1104.381,A -85,B 0,C 180,E1 30133.208,E2 30133.208} C_VEL
LIN {X 0,Y 642.037,Z 1090.021,A -85,B 0,C 180,E1 30131.099,E2 30131.099} C_VEL
LIN {X 0,Y 642.839,Z 1076.848,A -85,B 0,C 180,E1 30129.419,E2 30129.419} C_VEL
LIN {X 0,Y 643.936,Z 1060.155,A -85,B 0,C 180,E1 30127.543,E2 30127.543} C_VEL
LIN {X 0,Y 645.033,Z 1044.316,A -85,B 0,C 180,E1 30125.989,E2 30125.989} C_VEL
LIN {X 0,Y 646.36,Z 1026.198,A -85,B 0,C 180,E1 30124.406,E2 30124.406} C_VEL
LIN {X 0,Y 647.746,Z 1007.052,A -85,B 0,C 180,E1 30122.96,E2 30122.96} C_VEL
LIN {X 0,Y 649.227,Z 987.158,A -85,B 0,C 180,E1 30121.632,E2 30121.632} C_VEL
LIN {X 0,Y 650.633,Z 966.296,A -85,B 0,C 180,E1 30120.439,E2 30120.439} C_VEL
LIN {X 0,Y 651.976,Z 946.21,A -85,B 0,C 180,E1 30119.443,E2 30119.443} C_VEL
LIN {X 0,Y 653.34,Z 923.085,A -85,B 0,C 180,E1 30118.48,E2 30118.48} C_VEL
LIN {X 0,Y 654.396,Z 902.76,A -85,B 0,C 180,E1 30117.774,E2 30117.774} C_VEL
LIN {X 0,Y 655.464,Z 879.536,A -85,B 0,C 180,E1 30117.11,E2 30117.11} C_VEL
LIN {X 0,Y 656.325,Z 855.541,A -85,B 0,C 180,E1 30116.602,E2 30116.602} C_VEL
LIN {X 0,Y 656.956,Z 830.856,A -85,B 0,C 180,E1 30116.223,E2 30116.223} C_VEL
LIN {X 0,Y 659.889,Z 593.27,A -85,B 0,C 180,E1 30113.302,E2 30113.302} C_VEL
LIN {X 0,Y 661.283,Z 479.099,A -85,B 0,C 180,E1 30111.868,E2 30111.868} C_VEL
LIN {X 0,Y 654.785,Z 450.939,A -85,B 0,C 180,E1 30111.012,E2 30111.012} C_VEL
LIN {X 0,Y 654.628,Z 448.513,A -85,B 0,C 180,E1 30110.82,E2 30110.82} C_VEL
LIN {X 0,Y 646.057,Z 425.931,A -85,B 0,C 180,E1 30108.377,E2 30108.377} C_VEL
LIN {X 0,Y 640.832,Z 412.593,A -85,B 0,C 180,E1 30106.822,E2 30106.822} C_VEL
LIN {X 0,Y 640.806,Z 412.405,A -85,B 0,C 180,E1 30103.853,E2 30103.853} C_VEL
LIN {X 0,Y 640.799,Z 412.367,A -85,B 0,C 180,E1 30100.593,E2 30100.593} C_VEL
LIN {X 0,Y 640.826,Z 412.401,A -85,B 0,C 180,E1 30097.567,E2 30097.567} C_VEL
LIN {X 0,Y 640.802,Z 412.408,A -85,B 0,C 180,E1 30094.367,E2 30094.367} C_VEL
LIN {X 0,Y 640.827,Z 412.411,A -85,B 0,C 180,E1 30091.305,E2 30091.305} C_VEL
LIN {X 0,Y 640.806,Z 412.391,A -85,B 0,C 180,E1 30088.216,E2 30088.216} C_VEL
LIN {X 0,Y 640.821,Z 412.396,A -85,B 0,C 180,E1 30085.178,E2 30085.178} C_VEL
LIN {X 0,Y 640.809,Z 412.403,A -85,B 0,C 180,E1 30082.05,E2 30082.05} C_VEL
LIN {X 0,Y 640.813,Z 412.394,A -85,B 0,C 180,E1 30078.99,E2 30078.99} C_VEL
LIN {X 0,Y 640.814,Z 412.405,A -85,B 0,C 180,E1 30075.939,E2 30075.939} C_VEL
LIN {X 0,Y 640.809,Z 412.405,A -85,B 0,C 180,E1 30072.893,E2 30072.893} C_VEL
LIN {X 0,Y 640.819,Z 412.403,A -85,B 0,C 180,E1 30069.792,E2 30069.792} C_VEL
LIN {X 0,Y 640.804,Z 412.406,A -85,B 0,C 180,E1 30066.721,E2 30066.721} C_VEL
LIN {X 0,Y 640.822,Z 412.394,A -85,B 0,C 180,E1 30063.668,E2 30063.668} C_VEL
LIN {X 0,Y 640.796,Z 412.407,A -85,B 0,C 180,E1 30060.626,E2 30060.626} C_VEL
LIN {X 0,Y 640.825,Z 412.39,A -85,B 0,C 180,E1 30057.585,E2 30057.585} C_VEL
LIN {X 0,Y 640.79,Z 412.407,A -85,B 0,C 180,E1 30054.538,E2 30054.538} C_VEL
LIN {X 0,Y 640.828,Z 412.388,A -85,B 0,C 180,E1 30051.476,E2 30051.476} C_VEL
LIN {X 0,Y 640.783,Z 412.406,A -85,B 0,C 180,E1 30048.479,E2 30048.479} C_VEL
LIN {X 0,Y 640.831,Z 412.39,A -85,B 0,C 180,E1 30045.451,E2 30045.451} C_VEL
LIN {X 0,Y 640.777,Z 412.402,A -85,B 0,C 180,E1 30042.445,E2 30042.445} C_VEL
LIN {X 0,Y 640.834,Z 412.398,A -85,B 0,C 180,E1 30039.42,E2 30039.42} C_VEL
LIN {X 0,Y 640.769,Z 412.392,A -85,B 0,C 180,E1 30036.454,E2 30036.454} C_VEL
LIN {X 0,Y 640.805,Z 412.406,A -85,B 0,C 180,E1 30033.593,E2 30033.593} C_VEL
LIN {X 0,Y 640.769,Z 412.409,A -85,B 0,C 180,E1 30030.455,E2 30030.455} C_VEL
LIN {X 0,Y 640.771,Z 412.405,A -85,B 0,C 180,E1 30027.746,E2 30027.746} C_VEL
LIN {X 0,Y 640.769,Z 412.409,A -85,B 0,C 180,E1 30024.515,E2 30024.515} C_VEL
LIN {X 0,Y 640.753,Z 412.411,A -85,B 0,C 180,E1 30021.833,E2 30021.833} C_VEL
LIN {X 0,Y 640.803,Z 412.365,A -85,B 0,C 180,E1 30018.816,E2 30018.816} C_VEL
LIN {X 0,Y 640.739,Z 412.407,A -85,B 0,C 180,E1 30015.893,E2 30015.893} C_VEL
LIN {X 0,Y 640.759,Z 412.412,A -85,B 0,C 180,E1 30014.409,E2 30014.409} C_VEL
LIN {X 0,Y 639.719,Z 412.531,A -85,B 0,C 180,E1 30013.72,E2 30013.72} C_VEL
LIN {X 0,Y 633.311,Z 413.288,A -85,B 0,C 180,E1 30011.789,E2 30011.789} C_VEL
LIN {X 0,Y 632.822,Z 413.352,A -85,B 0,C 180,E1 30011.287,E2 30011.287} C_VEL
LIN {X 0,Y 632.794,Z 413.381,A -85,B 0,C 180,E1 30008.158,E2 30008.158} C_VEL
LIN {X 0,Y 632.849,Z 413.806,A -85,B 0,C 180,E1 30007.752,E2 30007.752} C_VEL
LIN {X 0,Y 634.067,Z 416.827,A -85,B 0,C 180,E1 30007.402,E2 30007.402} C_VEL
LIN {X 0,Y 650.137,Z 442.775,A -85,B 0,C 180,E1 30005.854,E2 30005.854} C_VEL
LIN {X 0,Y 655.244,Z 451.774,A -85,B 0,C 180,E1 30005.372,E2 30005.372} C_VEL
LIN {X 0,Y 651.622,Z 700.546,A -85,B 0,C 180,E1 30002.253,E2 30002.253} C_VEL
LIN {X 0,Y 650.1,Z 804.715,A -85,B 0,C 180,E1 30000.944,E2 30000.944} C_VEL
LIN {X 0,Y 649.266,Z 829.906,A -85,B 0,C 180,E1 30000.471,E2 30000.471} C_VEL
LIN {X 0,Y 648.355,Z 850.272,A -85,B 0,C 180,E1 29999.959,E2 29999.959} C_VEL
LIN {X 0,Y 647.239,Z 872.307,A -85,B 0,C 180,E1 29999.272,E2 29999.272} C_VEL
LIN {X 0,Y 645.751,Z 895.151,A -85,B 0,C 180,E1 29998.383,E2 29998.383} C_VEL
LIN {X 0,Y 644.342,Z 916.563,A -85,B 0,C 180,E1 29997.394,E2 29997.394} C_VEL
LIN {X 0,Y 642.676,Z 938.508,A -85,B 0,C 180,E1 29996.193,E2 29996.193} C_VEL
LIN {X 0,Y 640.948,Z 960.786,A -85,B 0,C 180,E1 29994.778,E2 29994.778} C_VEL
LIN {X 0,Y 639.435,Z 979.714,A -85,B 0,C 180,E1 29993.379,E2 29993.379} C_VEL
LIN {X 0,Y 637.994,Z 998.033,A -85,B 0,C 180,E1 29991.853,E2 29991.853} C_VEL
LIN {X 0,Y 636.674,Z 1015.124,A -85,B 0,C 180,E1 29990.213,E2 29990.213} C_VEL
LIN {X 0,Y 635.543,Z 1030.701,A -85,B 0,C 180,E1 29988.53,E2 29988.53} C_VEL
LIN {X 0,Y 634.483,Z 1046.475,A -85,B 0,C 180,E1 29986.573,E2 29986.573} C_VEL
LIN {X 0,Y 633.678,Z 1059.69,A -85,B 0,C 180,E1 29984.7,E2 29984.7} C_VEL
LIN {X 0,Y 633.011,Z 1072.476,A -85,B 0,C 180,E1 29982.591,E2 29982.591} C_VEL
LIN {X 0,Y 632.586,Z 1082.543,A -85,B 0,C 180,E1 29980.657,E2 29980.657} C_VEL
LIN {X 0,Y 632.252,Z 1092.154,A -85,B 0,C 180,E1 29978.458,E2 29978.458} C_VEL
LIN {X 0,Y 632.07,Z 1099.038,A -85,B 0,C 180,E1 29976.54,E2 29976.54} C_VEL
LIN {X 0,Y 631.966,Z 1105.363,A -85,B 0,C 180,E1 29974.356,E2 29974.356} C_VEL
LIN {X 0,Y 631.925,Z 1109.732,A -85,B 0,C 180,E1 29972.267,E2 29972.267} C_VEL
LIN {X 0,Y 631.924,Z 1112.622,A -85,B 0,C 180,E1 29970.272,E2 29970.272} C_VEL
LIN {X 0,Y 631.908,Z 1114.269,A -85,B 0,C 180,E1 29967.914,E2 29967.914} C_VEL
LIN {X 0,Y 631.905,Z 1114.272,A -85,B 0,C 180,E1 29966.008,E2 29966.008} C_VEL
LIN {X 0,Y 631.92,Z 1112.74,A -85,B 0,C 180,E1 29963.732,E2 29963.732} C_VEL
LIN {X 0,Y 631.93,Z 1109.87,A -85,B 0,C 180,E1 29961.721,E2 29961.721} C_VEL
LIN {X 0,Y 631.97,Z 1105.694,A -85,B 0,C 180,E1 29959.701,E2 29959.701} C_VEL
LIN {X 0,Y 632.07,Z 1099.261,A -85,B 0,C 180,E1 29957.437,E2 29957.437} C_VEL
LIN {X 0,Y 632.238,Z 1092.452,A -85,B 0,C 180,E1 29955.53,E2 29955.53} C_VEL
LIN {X 0,Y 632.575,Z 1082.683,A -85,B 0,C 180,E1 29953.281,E2 29953.281} C_VEL
LIN {X 0,Y 632.99,Z 1072.881,A -85,B 0,C 180,E1 29951.392,E2 29951.392} C_VEL
LIN {X 0,Y 633.638,Z 1060.655,A -85,B 0,C 180,E1 29949.353,E2 29949.353} C_VEL
LIN {X 0,Y 634.421,Z 1047.36,A -85,B 0,C 180,E1 29947.455,E2 29947.455} C_VEL
LIN {X 0,Y 635.446,Z 1032.255,A -85,B 0,C 180,E1 29945.554,E2 29945.554} C_VEL
LIN {X 0,Y 636.591,Z 1016.212,A -85,B 0,C 180,E1 29943.809,E2 29943.809} C_VEL
LIN {X 0,Y 637.938,Z 998.859,A -85,B 0,C 180,E1 29942.13,E2 29942.13} C_VEL
LIN {X 0,Y 639.387,Z 980.355,A -85,B 0,C 180,E1 29940.582,E2 29940.582} C_VEL
LIN {X 0,Y 640.905,Z 961.312,A -85,B 0,C 180,E1 29939.169,E2 29939.169} C_VEL
LIN {X 0,Y 642.64,Z 939.008,A -85,B 0,C 180,E1 29937.746,E2 29937.746} C_VEL
LIN {X 0,Y 644.342,Z 916.634,A -85,B 0,C 180,E1 29936.518,E2 29936.518} C_VEL
LIN {X 0,Y 645.745,Z 895.277,A -85,B 0,C 180,E1 29935.531,E2 29935.531} C_VEL
LIN {X 0,Y 647.196,Z 872.968,A -85,B 0,C 180,E1 29934.661,E2 29934.661} C_VEL
LIN {X 0,Y 648.373,Z 850.047,A -85,B 0,C 180,E1 29933.944,E2 29933.944} C_VEL
LIN {X 0,Y 649.283,Z 829.603,A -85,B 0,C 180,E1 29933.431,E2 29933.431} C_VEL
LIN {X 0,Y 650.112,Z 804.128,A -85,B 0,C 180,E1 29932.957,E2 29932.957} C_VEL
LIN {X 0,Y 652.978,Z 605.074,A -85,B 0,C 180,E1 29930.468,E2 29930.468} C_VEL
LIN {X 0,Y 655.125,Z 451.157,A -85,B 0,C 180,E1 29928.52,E2 29928.52} C_VEL
LIN {X 0,Y 642.562,Z 430.118,A -85,B 0,C 180,E1 29927.296,E2 29927.296} C_VEL
LIN {X 0,Y 633.8,Z 416.393,A -85,B 0,C 180,E1 29926.396,E2 29926.396} C_VEL
LIN {X 0,Y 632.809,Z 413.522,A -85,B 0,C 180,E1 29925.994,E2 29925.994} C_VEL
LIN {X 0,Y 632.875,Z 413.37,A -85,B 0,C 180,E1 29922.987,E2 29922.987} C_VEL
LIN {X 0,Y 632.801,Z 413.392,A -85,B 0,C 180,E1 29920.024,E2 29920.024} C_VEL
LIN {X 0,Y 632.833,Z 413.364,A -85,B 0,C 180,E1 29917.354,E2 29917.354} C_VEL
LIN {X 0,Y 632.823,Z 413.393,A -85,B 0,C 180,E1 29914.229,E2 29914.229} C_VEL
LIN {X 0,Y 632.822,Z 413.383,A -85,B 0,C 180,E1 29911.534,E2 29911.534} C_VEL
LIN {X 0,Y 632.848,Z 413.367,A -85,B 0,C 180,E1 29908.351,E2 29908.351} C_VEL
LIN {X 0,Y 632.828,Z 413.401,A -85,B 0,C 180,E1 29905.551,E2 29905.551} C_VEL
LIN {X 0,Y 632.882,Z 413.396,A -85,B 0,C 180,E1 29902.445,E2 29902.445} C_VEL
LIN {X 0,Y 632.835,Z 413.387,A -85,B 0,C 180,E1 29899.474,E2 29899.474} C_VEL
LIN {X 0,Y 632.883,Z 413.378,A -85,B 0,C 180,E1 29896.333,E2 29896.333} C_VEL
LIN {X 0,Y 632.846,Z 413.399,A -85,B 0,C 180,E1 29893.337,E2 29893.337} C_VEL
LIN {X 0,Y 632.884,Z 413.391,A -85,B 0,C 180,E1 29890.173,E2 29890.173} C_VEL
LIN {X 0,Y 632.855,Z 413.388,A -85,B 0,C 180,E1 29887.149,E2 29887.149} C_VEL
LIN {X 0,Y 632.879,Z 413.391,A -85,B 0,C 180,E1 29883.986,E2 29883.986} C_VEL
LIN {X 0,Y 632.883,Z 413.385,A -85,B 0,C 180,E1 29880.815,E2 29880.815} C_VEL
LIN {X 0,Y 632.866,Z 413.38,A -85,B 0,C 180,E1 29877.646,E2 29877.646} C_VEL
LIN {X 0,Y 632.888,Z 413.394,A -85,B 0,C 180,E1 29874.561,E2 29874.561} C_VEL
LIN {X 0,Y 632.87,Z 413.385,A -85,B 0,C 180,E1 29871.459,E2 29871.459} C_VEL
LIN {X 0,Y 632.88,Z 413.38,A -85,B 0,C 180,E1 29868.333,E2 29868.333} C_VEL
LIN {X 0,Y 632.872,Z 413.395,A -85,B 0,C 180,E1 29865.222,E2 29865.222} C_VEL
LIN {X 0,Y 632.876,Z 413.395,A -85,B 0,C 180,E1 29862.151,E2 29862.151} C_VEL
LIN {X 0,Y 632.876,Z 413.382,A -85,B 0,C 180,E1 29859.025,E2 29859.025} C_VEL
LIN {X 0,Y 632.872,Z 413.396,A -85,B 0,C 180,E1 29855.944,E2 29855.944} C_VEL
LIN {X 0,Y 632.882,Z 413.375,A -85,B 0,C 180,E1 29852.809,E2 29852.809} C_VEL
LIN {X 0,Y 632.865,Z 413.388,A -85,B 0,C 180,E1 29849.735,E2 29849.735} C_VEL
LIN {X 0,Y 632.89,Z 413.399,A -85,B 0,C 180,E1 29846.531,E2 29846.531} C_VEL
LIN {X 0,Y 632.88,Z 413.392,A -85,B 0,C 180,E1 29843.33,E2 29843.33} C_VEL
LIN {X 0,Y 632.863,Z 413.388,A -85,B 0,C 180,E1 29840.099,E2 29840.099} C_VEL
LIN {X 0,Y 632.888,Z 413.381,A -85,B 0,C 180,E1 29837.012,E2 29837.012} C_VEL
LIN {X 0,Y 632.867,Z 413.517,A -85,B 0,C 180,E1 29833.908,E2 29833.908} C_VEL
LIN {X 0,Y 633.208,Z 414.975,A -85,B 0,C 180,E1 29833.679,E2 29833.679} C_VEL
LIN {X 0,Y 638.654,Z 428.018,A -85,B 0,C 180,E1 29832.074,E2 29832.074} C_VEL
LIN {X 0,Y 645.903,Z 447.063,A -85,B 0,C 180,E1 29829.909,E2 29829.909} C_VEL
LIN {X 0,Y 647.521,Z 451.218,A -85,B 0,C 180,E1 29829.496,E2 29829.496} C_VEL
LIN {X 0,Y 648.79,Z 454.293,A -85,B 0,C 180,E1 29829.351,E2 29829.351} C_VEL
LIN {X 0,Y 655.097,Z 482.382,A -85,B 0,C 180,E1 29828.509,E2 29828.509} C_VEL
LIN {X 0,Y 651.671,Z 724.648,A -85,B 0,C 180,E1 29825.477,E2 29825.477} C_VEL
LIN {X 0,Y 650.003,Z 842.909,A -85,B 0,C 180,E1 29823.997,E2 29823.997} C_VEL
LIN {X 0,Y 649.14,Z 868.477,A -85,B 0,C 180,E1 29823.522,E2 29823.522} C_VEL
LIN {X 0,Y 648.228,Z 888.766,A -85,B 0,C 180,E1 29823.017,E2 29823.017} C_VEL
LIN {X 0,Y 647.099,Z 911.365,A -85,B 0,C 180,E1 29822.319,E2 29822.319} C_VEL
LIN {X 0,Y 645.623,Z 934.643,A -85,B 0,C 180,E1 29821.422,E2 29821.422} C_VEL
LIN {X 0,Y 644.216,Z 957.044,A -85,B 0,C 180,E1 29820.397,E2 29820.397} C_VEL
LIN {X 0,Y 642.597,Z 979.04,A -85,B 0,C 180,E1 29819.199,E2 29819.199} C_VEL
LIN {X 0,Y 641.169,Z 997.633,A -85,B 0,C 180,E1 29818.034,E2 29818.034} C_VEL
LIN {X 0,Y 639.571,Z 1017.994,A -85,B 0,C 180,E1 29816.56,E2 29816.56} C_VEL
LIN {X 0,Y 638.246,Z 1034.838,A -85,B 0,C 180,E1 29815.172,E2 29815.172} C_VEL
LIN {X 0,Y 636.789,Z 1053.673,A -85,B 0,C 180,E1 29813.407,E2 29813.407} C_VEL
LIN {X 0,Y 635.68,Z 1068.779,A -85,B 0,C 180,E1 29811.791,E2 29811.791} C_VEL
LIN {X 0,Y 634.579,Z 1085.115,A -85,B 0,C 180,E1 29809.802,E2 29809.802} C_VEL
LIN {X 0,Y 633.767,Z 1097.88,A -85,B 0,C 180,E1 29808.013,E2 29808.013} C_VEL
LIN {X 0,Y 633.094,Z 1110.73,A -85,B 0,C 180,E1 29805.951,E2 29805.951} C_VEL
LIN {X 0,Y 632.626,Z 1121.101,A -85,B 0,C 180,E1 29803.994,E2 29803.994} C_VEL
LIN {X 0,Y 632.301,Z 1130.77,A -85,B 0,C 180,E1 29801.863,E2 29801.863} C_VEL
LIN {X 0,Y 632.082,Z 1138.21,A -85,B 0,C 180,E1 29799.837,E2 29799.837} C_VEL
LIN {X 0,Y 631.971,Z 1143.999,A -85,B 0,C 180,E1 29797.912,E2 29797.912} C_VEL
LIN {X 0,Y 631.917,Z 1149.176,A -85,B 0,C 180,E1 29795.63,E2 29795.63} C_VEL
LIN {X 0,Y 631.914,Z 1152.124,A -85,B 0,C 180,E1 29793.72,E2 29793.72} C_VEL
LIN {X 0,Y 631.898,Z 1154.103,A -85,B 0,C 180,E1 29791.541,E2 29791.541} C_VEL
LIN {X 0,Y 631.884,Z 1154.373,A -85,B 0,C 180,E1 29789.456,E2 29789.456} C_VEL
LIN {X 0,Y 631.901,Z 1153.428,A -85,B 0,C 180,E1 29787.551,E2 29787.551} C_VEL
LIN {X 0,Y 631.914,Z 1150.768,A -85,B 0,C 180,E1 29785.28,E2 29785.28} C_VEL
LIN {X 0,Y 631.947,Z 1146.896,A -85,B 0,C 180,E1 29783.276,E2 29783.276} C_VEL
LIN {X 0,Y 632.009,Z 1141.71,A -85,B 0,C 180,E1 29781.264,E2 29781.264} C_VEL
LIN {X 0,Y 632.176,Z 1134.308,A -85,B 0,C 180,E1 29779.059,E2 29779.059} C_VEL
LIN {X 0,Y 632.442,Z 1126.345,A -85,B 0,C 180,E1 29777.119,E2 29777.119} C_VEL
LIN {X 0,Y 632.892,Z 1115.236,A -85,B 0,C 180,E1 29774.864,E2 29774.864} C_VEL
LIN {X 0,Y 633.409,Z 1104.544,A -85,B 0,C 180,E1 29773.02,E2 29773.02} C_VEL
LIN {X 0,Y 634.202,Z 1090.72,A -85,B 0,C 180,E1 29770.952,E2 29770.952} C_VEL
LIN {X 0,Y 635.115,Z 1076.846,A -85,B 0,C 180,E1 29769.157,E2 29769.157} C_VEL
LIN {X 0,Y 636.309,Z 1060.154,A -85,B 0,C 180,E1 29767.259,E2 29767.259} C_VEL
LIN {X 0,Y 637.506,Z 1044.255,A -85,B 0,C 180,E1 29765.681,E2 29765.681} C_VEL
LIN {X 0,Y 638.96,Z 1025.759,A -85,B 0,C 180,E1 29764.052,E2 29764.052} C_VEL
LIN {X 0,Y 640.433,Z 1007.056,A -85,B 0,C 180,E1 29762.626,E2 29762.626} C_VEL
LIN {X 0,Y 642.047,Z 986.745,A -85,B 0,C 180,E1 29761.258,E2 29761.258} C_VEL
LIN {X 0,Y 643.515,Z 966.192,A -85,B 0,C 180,E1 29760.081,E2 29760.081} C_VEL
LIN {X 0,Y 644.943,Z 945.919,A -85,B 0,C 180,E1 29759.073,E2 29759.073} C_VEL
LIN {X 0,Y 646.422,Z 922.455,A -85,B 0,C 180,E1 29758.089,E2 29758.089} C_VEL
LIN {X 0,Y 647.572,Z 901.724,A -85,B 0,C 180,E1 29757.366,E2 29757.366} C_VEL
LIN {X 0,Y 648.742,Z 877.53,A -85,B 0,C 180,E1 29756.682,E2 29756.682} C_VEL
LIN {X 0,Y 649.64,Z 854.777,A -85,B 0,C 180,E1 29756.203,E2 29756.203} C_VEL
LIN {X 0,Y 650.299,Z 829.815,A -85,B 0,C 180,E1 29755.82,E2 29755.82} C_VEL
LIN {X 0,Y 653.455,Z 593.128,A -85,B 0,C 180,E1 29752.883,E2 29752.883} C_VEL
LIN {X 0,Y 654.934,Z 480.882,A -85,B 0,C 180,E1 29751.459,E2 29751.459} C_VEL
LIN {X 0,Y 648.066,Z 452.372,A -85,B 0,C 180,E1 29750.588,E2 29750.588} C_VEL
LIN {X 0,Y 646.886,Z 449.826,A -85,B 0,C 180,E1 29750.402,E2 29750.402} C_VEL
LIN {X 0,Y 639.026,Z 429.301,A -85,B 0,C 180,E1 29748.142,E2 29748.142} C_VEL
LIN {X 0,Y 632.873,Z 413.588,A -85,B 0,C 180,E1 29746.283,E2 29746.283} C_VEL
LIN {X 0,Y 632.888,Z 413.368,A -85,B 0,C 180,E1 29743.289,E2 29743.289} C_VEL
LIN {X 0,Y 632.849,Z 413.363,A -85,B 0,C 180,E1 29740.257,E2 29740.257} C_VEL
LIN {X 0,Y 632.887,Z 413.383,A -85,B 0,C 180,E1 29737.225,E2 29737.225} C_VEL
LIN {X 0,Y 632.86,Z 413.399,A -85,B 0,C 180,E1 29734.116,E2 29734.116} C_VEL
LIN {X 0,Y 632.886,Z 413.396,A -85,B 0,C 180,E1 29731.001,E2 29731.001} C_VEL
LIN {X 0,Y 632.867,Z 413.383,A -85,B 0,C 180,E1 29727.883,E2 29727.883} C_VEL
LIN {X 0,Y 632.887,Z 413.378,A -85,B 0,C 180,E1 29724.709,E2 29724.709} C_VEL
LIN {X 0,Y 632.891,Z 413.399,A -85,B 0,C 180,E1 29721.479,E2 29721.479} C_VEL
LIN {X 0,Y 632.883,Z 413.382,A -85,B 0,C 180,E1 29718.229,E2 29718.229} C_VEL
LIN {X 0,Y 632.877,Z 413.384,A -85,B 0,C 180,E1 29715.111,E2 29715.111} C_VEL
LIN {X 0,Y 632.881,Z 413.391,A -85,B 0,C 180,E1 29711.945,E2 29711.945} C_VEL
LIN {X 0,Y 632.864,Z 413.378,A -85,B 0,C 180,E1 29708.816,E2 29708.816} C_VEL
LIN {X 0,Y 632.884,Z 413.393,A -85,B 0,C 180,E1 29705.803,E2 29705.803} C_VEL
LIN {X 0,Y 632.859,Z 413.384,A -85,B 0,C 180,E1 29702.717,E2 29702.717} C_VEL
LIN {X 0,Y 632.887,Z 413.395,A -85,B 0,C 180,E1 29699.638,E2 29699.638} C_VEL
LIN {X 0,Y 632.853,Z 413.389,A -85,B 0,C 180,E1 29696.558,E2 29696.558} C_VEL
LIN {X 0,Y 632.891,Z 413.393,A -85,B 0,C 180,E1 29693.468,E2 29693.468} C_VEL
LIN {X 0,Y 632.847,Z 413.393,A -85,B 0,C 180,E1 29690.45,E2 29690.45} C_VEL
LIN {X 0,Y 632.892,Z 413.384,A -85,B 0,C 180,E1 29687.314,E2 29687.314} C_VEL
LIN {X 0,Y 632.84,Z 413.396,A -85,B 0,C 180,E1 29684.325,E2 29684.325} C_VEL
LIN {X 0,Y 632.893,Z 413.38,A -85,B 0,C 180,E1 29681.294,E2 29681.294} C_VEL
LIN {X 0,Y 632.831,Z 413.397,A -85,B 0,C 180,E1 29678.289,E2 29678.289} C_VEL
LIN {X 0,Y 632.894,Z 413.378,A -85,B 0,C 180,E1 29675.249,E2 29675.249} C_VEL
LIN {X 0,Y 632.823,Z 413.39,A -85,B 0,C 180,E1 29672.217,E2 29672.217} C_VEL
LIN {X 0,Y 632.897,Z 413.395,A -85,B 0,C 180,E1 29669.211,E2 29669.211} C_VEL
LIN {X 0,Y 632.816,Z 413.398,A -85,B 0,C 180,E1 29666.208,E2 29666.208} C_VEL
LIN {X 0,Y 632.864,Z 413.387,A -85,B 0,C 180,E1 29663.329,E2 29663.329} C_VEL
LIN {X 0,Y 632.813,Z 413.395,A -85,B 0,C 180,E1 29660.309,E2 29660.309} C_VEL
LIN {X 0,Y 632.805,Z 413.347,A -85,B 0,C 180,E1 29657.688,E2 29657.688} C_VEL
LIN {X 0,Y 632.836,Z 413.401,A -85,B 0,C 180,E1 29654.55,E2 29654.55} C_VEL
LIN {X 0,Y 632.789,Z 413.351,A -85,B 0,C 180,E1 29651.77,E2 29651.77} C_VEL
LIN {X 0,Y 632.822,Z 413.352,A -85,B 0,C 180,E1 29651.287,E2 29651.287} C_VEL
LIN {X 0,Y 631.838,Z 413.488,A -85,B 0,C 180,E1 29650.822,E2 29650.822} C_VEL
LIN {X 0,Y 625.622,Z 414.304,A -85,B 0,C 180,E1 29649.632,E2 29649.632} C_VEL
LIN {X 0,Y 624.888,Z 414.391,A -85,B 0,C 180,E1 29649.225,E2 29649.225} C_VEL
LIN {X 0,Y 624.914,Z 414.684,A -85,B 0,C 180,E1 29648.318,E2 29648.318} C_VEL
LIN {X 0,Y 625.738,Z 417.163,A -85,B 0,C 180,E1 29648.039,E2 29648.039} C_VEL
LIN {X 0,Y 635.654,Z 432.716,A -85,B 0,C 180,E1 29647.049,E2 29647.049} C_VEL
LIN {X 0,Y 646.97,Z 451.218,A -85,B 0,C 180,E1 29645.961,E2 29645.961} C_VEL
LIN {X 0,Y 648.918,Z 454.861,A -85,B 0,C 180,E1 29645.772,E2 29645.772} C_VEL
LIN {X 0,Y 645.073,Z 703.417,A -85,B 0,C 180,E1 29642.631,E2 29642.631} C_VEL
LIN {X 0,Y 643.478,Z 804.994,A -85,B 0,C 180,E1 29641.342,E2 29641.342} C_VEL
LIN {X 0,Y 642.596,Z 830.254,A -85,B 0,C 180,E1 29640.864,E2 29640.864} C_VEL
LIN {X 0,Y 641.638,Z 850.502,A -85,B 0,C 180,E1 29640.351,E2 29640.351} C_VEL
LIN {X 0,Y 640.421,Z 873.054,A -85,B 0,C 180,E1 29639.64,E2 29639.64} C_VEL
LIN {X 0,Y 638.881,Z 895.271,A -85,B 0,C 180,E1 29638.768,E2 29638.768} C_VEL
LIN {X 0,Y 637.309,Z 917.677,A -85,B 0,C 180,E1 29637.722,E2 29637.722} C_VEL
LIN {X 0,Y 635.566,Z 938.933,A -85,B 0,C 180,E1 29636.539,E2 29636.539} C_VEL
LIN {X 0,Y 633.976,Z 957.616,A -85,B 0,C 180,E1 29635.348,E2 29635.348} C_VEL
LIN {X 0,Y 632.2,Z 978.183,A -85,B 0,C 180,E1 29633.835,E2 29633.835} C_VEL
LIN {X 0,Y 630.707,Z 995.784,A -85,B 0,C 180,E1 29632.364,E2 29632.364} C_VEL
LIN {X 0,Y 629.134,Z 1014.612,A -85,B 0,C 180,E1 29630.563,E2 29630.563} C_VEL
LIN {X 0,Y 627.966,Z 1029.458,A -85,B 0,C 180,E1 29628.948,E2 29628.948} C_VEL
LIN {X 0,Y 626.742,Z 1046.085,A -85,B 0,C 180,E1 29626.88,E2 29626.88} C_VEL
LIN {X 0,Y 625.901,Z 1058.595,A -85,B 0,C 180,E1 29625.094,E2 29625.094} C_VEL
LIN {X 0,Y 625.135,Z 1072.188,A -85,B 0,C 180,E1 29622.846,E2 29622.846} C_VEL
LIN {X 0,Y 624.68,Z 1081.831,A -85,B 0,C 180,E1 29620.981,E2 29620.981} C_VEL
LIN {X 0,Y 624.314,Z 1091.603,A -85,B 0,C 180,E1 29618.752,E2 29618.752} C_VEL
LIN {X 0,Y 624.086,Z 1098.565,A -85,B 0,C 180,E1 29616.809,E2 29616.809} C_VEL
LIN {X 0,Y 623.977,Z 1104.519,A -85,B 0,C 180,E1 29614.78,E2 29614.78} C_VEL
LIN {X 0,Y 623.93,Z 1109.481,A -85,B 0,C 180,E1 29612.48,E2 29612.48} C_VEL
LIN {X 0,Y 623.907,Z 1112.333,A -85,B 0,C 180,E1 29610.551,E2 29610.551} C_VEL
LIN {X 0,Y 623.892,Z 1114.165,A -85,B 0,C 180,E1 29608.347,E2 29608.347} C_VEL
LIN {X 0,Y 623.891,Z 1114.353,A -85,B 0,C 180,E1 29606.324,E2 29606.324} C_VEL
LIN {X 0,Y 623.906,Z 1113.365,A -85,B 0,C 180,E1 29604.39,E2 29604.39} C_VEL
LIN {X 0,Y 623.927,Z 1110.561,A -85,B 0,C 180,E1 29602.054,E2 29602.054} C_VEL
LIN {X 0,Y 623.952,Z 1106.647,A -85,B 0,C 180,E1 29600.034,E2 29600.034} C_VEL
LIN {X 0,Y 624.035,Z 1101.097,A -85,B 0,C 180,E1 29597.883,E2 29597.883} C_VEL
LIN {X 0,Y 624.225,Z 1093.728,A -85,B 0,C 180,E1 29595.719,E2 29595.719} C_VEL
LIN {X 0,Y 624.507,Z 1085.983,A -85,B 0,C 180,E1 29593.824,E2 29593.824} C_VEL
LIN {X 0,Y 625.003,Z 1074.743,A -85,B 0,C 180,E1 29591.533,E2 29591.533} C_VEL
LIN {X 0,Y 625.567,Z 1064.24,A -85,B 0,C 180,E1 29589.705,E2 29589.705} C_VEL
LIN {X 0,Y 626.479,Z 1049.798,A -85,B 0,C 180,E1 29587.536,E2 29587.536} C_VEL
LIN {X 0,Y 627.427,Z 1036.665,A -85,B 0,C 180,E1 29585.822,E2 29585.822} C_VEL
LIN {X 0,Y 628.708,Z 1020.055,A -85,B 0,C 180,E1 29583.912,E2 29583.912} C_VEL
LIN {X 0,Y 630.024,Z 1003.854,A -85,B 0,C 180,E1 29582.289,E2 29582.289} C_VEL
LIN {X 0,Y 631.585,Z 985.487,A -85,B 0,C 180,E1 29580.657,E2 29580.657} C_VEL
LIN {X 0,Y 633.288,Z 965.582,A -85,B 0,C 180,E1 29579.127,E2 29579.127} C_VEL
LIN {X 0,Y 635.054,Z 945.099,A -85,B 0,C 180,E1 29577.74,E2 29577.74} C_VEL
LIN {X 0,Y 636.661,Z 925.417,A -85,B 0,C 180,E1 29576.601,E2 29576.601} C_VEL
LIN {X 0,Y 638.355,Z 903.742,A -85,B 0,C 180,E1 29575.511,E2 29575.511} C_VEL
LIN {X 0,Y 639.874,Z 881.028,A -85,B 0,C 180,E1 29574.568,E2 29574.568} C_VEL
LIN {X 0,Y 641.252,Z 858.076,A -85,B 0,C 180,E1 29573.774,E2 29573.774} C_VEL
LIN {X 0,Y 642.398,Z 834.518,A -85,B 0,C 180,E1 29573.143,E2 29573.143} C_VEL
LIN {X 0,Y 643.26,Z 812.813,A -85,B 0,C 180,E1 29572.697,E2 29572.697} C_VEL
LIN {X 0,Y 643.943,Z 780.348,A -85,B 0,C 180,E1 29572.238,E2 29572.238} C_VEL
LIN {X 0,Y 647.701,Z 532.313,A -85,B 0,C 180,E1 29569.121,E2 29569.121} C_VEL
LIN {X 0,Y 648.894,Z 454.337,A -85,B 0,C 180,E1 29568.114,E2 29568.114} C_VEL
LIN {X 0,Y 637.397,Z 435.13,A -85,B 0,C 180,E1 29566.972,E2 29566.972} C_VEL
LIN {X 0,Y 628.438,Z 421.243,A -85,B 0,C 180,E1 29566.051,E2 29566.051} C_VEL
LIN {X 0,Y 625.457,Z 416.571,A -85,B 0,C 180,E1 29565.703,E2 29565.703} C_VEL
LIN {X 0,Y 624.909,Z 414.5,A -85,B 0,C 180,E1 29565.4,E2 29565.4} C_VEL
LIN {X 0,Y 624.861,Z 414.349,A -85,B 0,C 180,E1 29562.228,E2 29562.228} C_VEL
LIN {X 0,Y 624.881,Z 414.387,A -85,B 0,C 180,E1 29559.532,E2 29559.532} C_VEL
LIN {X 0,Y 624.875,Z 414.336,A -85,B 0,C 180,E1 29556.247,E2 29556.247} C_VEL
LIN {X 0,Y 624.885,Z 414.388,A -85,B 0,C 180,E1 29553.507,E2 29553.507} C_VEL
LIN {X 0,Y 624.889,Z 414.337,A -85,B 0,C 180,E1 29550.224,E2 29550.224} C_VEL
LIN {X 0,Y 624.893,Z 414.375,A -85,B 0,C 180,E1 29547.441,E2 29547.441} C_VEL
LIN {X 0,Y 624.907,Z 414.373,A -85,B 0,C 180,E1 29544.181,E2 29544.181} C_VEL
LIN {X 0,Y 624.901,Z 414.39,A -85,B 0,C 180,E1 29541.369,E2 29541.369} C_VEL
LIN {X 0,Y 624.92,Z 414.385,A -85,B 0,C 180,E1 29538.117,E2 29538.117} C_VEL
LIN {X 0,Y 624.91,Z 414.373,A -85,B 0,C 180,E1 29535.213,E2 29535.213} C_VEL
LIN {X 0,Y 624.916,Z 414.373,A -85,B 0,C 180,E1 29531.912,E2 29531.912} C_VEL
LIN {X 0,Y 624.947,Z 414.388,A -85,B 0,C 180,E1 29528.835,E2 29528.835} C_VEL
LIN {X 0,Y 624.916,Z 414.377,A -85,B 0,C 180,E1 29525.693,E2 29525.693} C_VEL
LIN {X 0,Y 624.947,Z 414.369,A -85,B 0,C 180,E1 29522.659,E2 29522.659} C_VEL
LIN {X 0,Y 624.921,Z 414.382,A -85,B 0,C 180,E1 29519.542,E2 29519.542} C_VEL
LIN {X 0,Y 624.946,Z 414.373,A -85,B 0,C 180,E1 29516.422,E2 29516.422} C_VEL
LIN {X 0,Y 624.924,Z 414.378,A -85,B 0,C 180,E1 29513.292,E2 29513.292} C_VEL
LIN {X 0,Y 624.943,Z 414.383,A -85,B 0,C 180,E1 29510.236,E2 29510.236} C_VEL
LIN {X 0,Y 624.931,Z 414.37,A -85,B 0,C 180,E1 29507.056,E2 29507.056} C_VEL
LIN {X 0,Y 624.938,Z 414.372,A -85,B 0,C 180,E1 29504.026,E2 29504.026} C_VEL
LIN {X 0,Y 624.942,Z 414.387,A -85,B 0,C 180,E1 29500.853,E2 29500.853} C_VEL
LIN {X 0,Y 624.946,Z 414.366,A -85,B 0,C 180,E1 29497.636,E2 29497.636} C_VEL
LIN {X 0,Y 624.943,Z 414.372,A -85,B 0,C 180,E1 29494.406,E2 29494.406} C_VEL
LIN {X 0,Y 624.951,Z 414.38,A -85,B 0,C 180,E1 29491.211,E2 29491.211} C_VEL
LIN {X 0,Y 624.927,Z 414.371,A -85,B 0,C 180,E1 29488.129,E2 29488.129} C_VEL
LIN {X 0,Y 624.95,Z 414.371,A -85,B 0,C 180,E1 29485.003,E2 29485.003} C_VEL
LIN {X 0,Y 624.916,Z 414.381,A -85,B 0,C 180,E1 29481.858,E2 29481.858} C_VEL
LIN {X 0,Y 624.953,Z 414.383,A -85,B 0,C 180,E1 29478.762,E2 29478.762} C_VEL
LIN {X 0,Y 624.911,Z 414.384,A -85,B 0,C 180,E1 29475.635,E2 29475.635} C_VEL
LIN {X 0,Y 624.987,Z 414.639,A -85,B 0,C 180,E1 29474.45,E2 29474.45} C_VEL
LIN {X 0,Y 632.371,Z 433.062,A -85,B 0,C 180,E1 29472.134,E2 29472.134} C_VEL
LIN {X 0,Y 639.103,Z 450.615,A -85,B 0,C 180,E1 29470.139,E2 29470.139} C_VEL
LIN {X 0,Y 642.999,Z 457.907,A -85,B 0,C 180,E1 29469.727,E2 29469.727} C_VEL
LIN {X 0,Y 648.823,Z 484.167,A -85,B 0,C 180,E1 29468.929,E2 29468.929} C_VEL
LIN {X 0,Y 645.13,Z 724.973,A -85,B 0,C 180,E1 29465.883,E2 29465.883} C_VEL
LIN {X 0,Y 643.344,Z 842.662,A -85,B 0,C 180,E1 29464.397,E2 29464.397} C_VEL
LIN {X 0,Y 642.421,Z 868.3,A -85,B 0,C 180,E1 29463.917,E2 29463.917} C_VEL
LIN {X 0,Y 641.453,Z 888.461,A -85,B 0,C 180,E1 29463.411,E2 29463.411} C_VEL
LIN {X 0,Y 640.244,Z 911.061,A -85,B 0,C 180,E1 29462.708,E2 29462.708} C_VEL
LIN {X 0,Y 638.679,Z 934.105,A -85,B 0,C 180,E1 29461.814,E2 29461.814} C_VEL
LIN {X 0,Y 637.204,Z 955.725,A -85,B 0,C 180,E1 29460.82,E2 29460.82} C_VEL
LIN {X 0,Y 635.551,Z 977.134,A -85,B 0,C 180,E1 29459.656,E2 29459.656} C_VEL
LIN {X 0,Y 634.047,Z 995.813,A -85,B 0,C 180,E1 29458.493,E2 29458.493} C_VEL
LIN {X 0,Y 632.281,Z 1017.138,A -85,B 0,C 180,E1 29456.962,E2 29456.962} C_VEL
LIN {X 0,Y 630.899,Z 1033.524,A -85,B 0,C 180,E1 29455.605,E2 29455.605} C_VEL
LIN {X 0,Y 629.373,Z 1051.819,A -85,B 0,C 180,E1 29453.899,E2 29453.899} C_VEL
LIN {X 0,Y 628.083,Z 1067.932,A -85,B 0,C 180,E1 29452.167,E2 29452.167} C_VEL
LIN {X 0,Y 626.916,Z 1083.704,A -85,B 0,C 180,E1 29450.249,E2 29450.249} C_VEL
LIN {X 0,Y 625.988,Z 1097.243,A -85,B 0,C 180,E1 29448.341,E2 29448.341} C_VEL
LIN {X 0,Y 625.277,Z 1109.688,A -85,B 0,C 180,E1 29446.347,E2 29446.347} C_VEL
LIN {X 0,Y 624.723,Z 1120.641,A -85,B 0,C 180,E1 29444.27,E2 29444.27} C_VEL
LIN {X 0,Y 624.359,Z 1129.99,A -85,B 0,C 180,E1 29442.204,E2 29442.204} C_VEL
LIN {X 0,Y 624.107,Z 1137.907,A -85,B 0,C 180,E1 29440.057,E2 29440.057} C_VEL
LIN {X 0,Y 623.995,Z 1143.745,A -85,B 0,C 180,E1 29438.106,E2 29438.106} C_VEL
LIN {X 0,Y 623.932,Z 1149.016,A -85,B 0,C 180,E1 29435.795,E2 29435.795} C_VEL
LIN {X 0,Y 623.914,Z 1152.124,A -85,B 0,C 180,E1 29433.767,E2 29433.767} C_VEL
LIN {X 0,Y 623.898,Z 1154.103,A -85,B 0,C 180,E1 29431.561,E2 29431.561} C_VEL
LIN {X 0,Y 623.884,Z 1154.373,A -85,B 0,C 180,E1 29429.449,E2 29429.449} C_VEL
LIN {X 0,Y 623.899,Z 1153.428,A -85,B 0,C 180,E1 29427.52,E2 29427.52} C_VEL
LIN {X 0,Y 623.912,Z 1150.769,A -85,B 0,C 180,E1 29425.22,E2 29425.22} C_VEL
LIN {X 0,Y 623.954,Z 1146.895,A -85,B 0,C 180,E1 29423.189,E2 29423.189} C_VEL
LIN {X 0,Y 624.02,Z 1141.71,A -85,B 0,C 180,E1 29421.151,E2 29421.151} C_VEL
LIN {X 0,Y 624.201,Z 1134.308,A -85,B 0,C 180,E1 29418.917,E2 29418.917} C_VEL
LIN {X 0,Y 624.477,Z 1126.75,A -85,B 0,C 180,E1 29417.046,E2 29417.046} C_VEL
LIN {X 0,Y 624.935,Z 1116.404,A -85,B 0,C 180,E1 29414.882,E2 29414.882} C_VEL
LIN {X 0,Y 625.519,Z 1105.115,A -85,B 0,C 180,E1 29412.895,E2 29412.895} C_VEL
LIN {X 0,Y 626.332,Z 1092.119,A -85,B 0,C 180,E1 29410.897,E2 29410.897} C_VEL
LIN {X 0,Y 627.346,Z 1077.615,A -85,B 0,C 180,E1 29408.985,E2 29408.985} C_VEL
LIN {X 0,Y 628.564,Z 1061.998,A -85,B 0,C 180,E1 29407.161,E2 29407.161} C_VEL
LIN {X 0,Y 629.943,Z 1044.821,A -85,B 0,C 180,E1 29405.426,E2 29405.426} C_VEL
LIN {X 0,Y 631.502,Z 1026.496,A -85,B 0,C 180,E1 29403.784,E2 29403.784} C_VEL
LIN {X 0,Y 633.078,Z 1007.684,A -85,B 0,C 180,E1 29402.332,E2 29402.332} C_VEL
LIN {X 0,Y 634.602,Z 989.134,A -85,B 0,C 180,E1 29401.072,E2 29401.072} C_VEL
LIN {X 0,Y 636.332,Z 966.899,A -85,B 0,C 180,E1 29399.766,E2 29399.766} C_VEL
LIN {X 0,Y 637.776,Z 947.653,A -85,B 0,C 180,E1 29398.792,E2 29398.792} C_VEL
LIN {X 0,Y 639.409,Z 924.062,A -85,B 0,C 180,E1 29397.775,E2 29397.775} C_VEL
LIN {X 0,Y 640.665,Z 902.921,A -85,B 0,C 180,E1 29397.023,E2 29397.023} C_VEL
LIN {X 0,Y 641.919,Z 879.445,A -85,B 0,C 180,E1 29396.338,E2 29396.338} C_VEL
LIN {X 0,Y 642.93,Z 855.423,A -85,B 0,C 180,E1 29395.821,E2 29395.821} C_VEL
LIN {X 0,Y 643.622,Z 831.617,A -85,B 0,C 180,E1 29395.446,E2 29395.446} C_VEL
LIN {X 0,Y 647.037,Z 594.351,A -85,B 0,C 180,E1 29392.472,E2 29392.472} C_VEL
LIN {X 0,Y 648.602,Z 482.67,A -85,B 0,C 180,E1 29391.046,E2 29391.046} C_VEL
LIN {X 0,Y 642.306,Z 456.369,A -85,B 0,C 180,E1 29390.231,E2 29390.231} C_VEL
LIN {X 0,Y 638.829,Z 450.206,A -85,B 0,C 180,E1 29389.864,E2 29389.864} C_VEL
LIN {X 0,Y 630.233,Z 427.869,A -85,B 0,C 180,E1 29387.355,E2 29387.355} C_VEL
LIN {X 0,Y 624.97,Z 414.615,A -85,B 0,C 180,E1 29385.739,E2 29385.739} C_VEL
LIN {X 0,Y 624.916,Z 414.335,A -85,B 0,C 180,E1 29382.596,E2 29382.596} C_VEL
LIN {X 0,Y 624.951,Z 414.364,A -85,B 0,C 180,E1 29379.54,E2 29379.54} C_VEL
LIN {X 0,Y 624.923,Z 414.371,A -85,B 0,C 180,E1 29376.408,E2 29376.408} C_VEL
LIN {X 0,Y 624.949,Z 414.37,A -85,B 0,C 180,E1 29373.284,E2 29373.284} C_VEL
LIN {X 0,Y 624.925,Z 414.386,A -85,B 0,C 180,E1 29370.159,E2 29370.159} C_VEL
LIN {X 0,Y 624.945,Z 414.387,A -85,B 0,C 180,E1 29367.129,E2 29367.129} C_VEL
LIN {X 0,Y 624.929,Z 414.366,A -85,B 0,C 180,E1 29363.979,E2 29363.979} C_VEL
LIN {X 0,Y 624.938,Z 414.38,A -85,B 0,C 180,E1 29360.904,E2 29360.904} C_VEL
LIN {X 0,Y 624.936,Z 414.376,A -85,B 0,C 180,E1 29357.794,E2 29357.794} C_VEL
LIN {X 0,Y 624.935,Z 414.366,A -85,B 0,C 180,E1 29354.643,E2 29354.643} C_VEL
LIN {X 0,Y 624.948,Z 414.387,A -85,B 0,C 180,E1 29351.443,E2 29351.443} C_VEL
LIN {X 0,Y 624.949,Z 414.363,A -85,B 0,C 180,E1 29348.187,E2 29348.187} C_VEL
LIN {X 0,Y 624.929,Z 414.379,A -85,B 0,C 180,E1 29344.957,E2 29344.957} C_VEL
LIN {X 0,Y 624.948,Z 414.371,A -85,B 0,C 180,E1 29341.834,E2 29341.834} C_VEL
LIN {X 0,Y 624.921,Z 414.375,A -85,B 0,C 180,E1 29338.808,E2 29338.808} C_VEL
LIN {X 0,Y 624.951,Z 414.375,A -85,B 0,C 180,E1 29335.687,E2 29335.687} C_VEL
LIN {X 0,Y 624.911,Z 414.369,A -85,B 0,C 180,E1 29332.646,E2 29332.646} C_VEL
LIN {X 0,Y 624.953,Z 414.38,A -85,B 0,C 180,E1 29329.584,E2 29329.584} C_VEL
LIN {X 0,Y 624.901,Z 414.367,A -85,B 0,C 180,E1 29326.49,E2 29326.49} C_VEL
LIN {X 0,Y 624.956,Z 414.384,A -85,B 0,C 180,E1 29323.409,E2 29323.409} C_VEL
LIN {X 0,Y 624.895,Z 414.379,A -85,B 0,C 180,E1 29320.365,E2 29320.365} C_VEL
LIN {X 0,Y 624.961,Z 414.377,A -85,B 0,C 180,E1 29317.32,E2 29317.32} C_VEL
LIN {X 0,Y 624.889,Z 414.387,A -85,B 0,C 180,E1 29314.272,E2 29314.272} C_VEL
LIN {X 0,Y 624.959,Z 414.367,A -85,B 0,C 180,E1 29311.211,E2 29311.211} C_VEL
LIN {X 0,Y 624.879,Z 414.384,A -85,B 0,C 180,E1 29308.176,E2 29308.176} C_VEL
LIN {X 0,Y 624.948,Z 414.386,A -85,B 0,C 180,E1 29305.163,E2 29305.163} C_VEL
LIN {X 0,Y 624.875,Z 414.39,A -85,B 0,C 180,E1 29302.203,E2 29302.203} C_VEL
LIN {X 0,Y 624.881,Z 414.366,A -85,B 0,C 180,E1 29299.605,E2 29299.605} C_VEL
LIN {X 0,Y 624.871,Z 414.358,A -85,B 0,C 180,E1 29296.325,E2 29296.325} C_VEL
LIN {X 0,Y 624.865,Z 414.37,A -85,B 0,C 180,E1 29293.605,E2 29293.605} C_VEL
LIN {X 0,Y 624.874,Z 414.361,A -85,B 0,C 180,E1 29290.388,E2 29290.388} C_VEL
LIN {X 0,Y 624.888,Z 414.391,A -85,B 0,C 180,E1 29289.225,E2 29289.225} C_VEL
LIN {X 0,Y 625.045,Z 415.334,A -85,B 0,C 180,E1 29288.85,E2 29288.85} C_VEL
LIN {X 0,Y 625.493,Z 418.366,A -85,B 0,C 180,E1 29288.446,E2 29288.446} C_VEL
LIN {X 0,Y 626.366,Z 423.477,A -85,B 0,C 180,E1 29288.061,E2 29288.061} C_VEL
LIN {X 0,Y 629.05,Z 433.928,A -85,B 0,C 180,E1 29287.548,E2 29287.548} C_VEL
LIN {X 0,Y 631.79,Z 439.799,A -85,B 0,C 180,E1 29287.239,E2 29287.239} C_VEL
LIN {X 0,Y 632.365,Z 440.676,A -85,B 0,C 180,E1 29287.183,E2 29287.183} C_VEL
LIN {X 0,Y 642.613,Z 457.797,A -85,B 0,C 180,E1 29286.18,E2 29286.18} C_VEL
LIN {X 0,Y 638.572,Z 704.813,A -85,B 0,C 180,E1 29283.035,E2 29283.035} C_VEL
LIN {X 0,Y 636.886,Z 805.378,A -85,B 0,C 180,E1 29281.747,E2 29281.747} C_VEL
LIN {X 0,Y 635.957,Z 830.601,A -85,B 0,C 180,E1 29281.265,E2 29281.265} C_VEL
LIN {X 0,Y 634.952,Z 850.731,A -85,B 0,C 180,E1 29280.751,E2 29280.751} C_VEL
LIN {X 0,Y 633.676,Z 873.135,A -85,B 0,C 180,E1 29280.04,E2 29280.04} C_VEL
LIN {X 0,Y 632.042,Z 895.42,A -85,B 0,C 180,E1 29279.159,E2 29279.159} C_VEL
LIN {X 0,Y 630.433,Z 916.765,A -85,B 0,C 180,E1 29278.158,E2 29278.158} C_VEL
LIN {X 0,Y 628.59,Z 938.316,A -85,B 0,C 180,E1 29276.959,E2 29276.959} C_VEL
LIN {X 0,Y 626.967,Z 956.286,A -85,B 0,C 180,E1 29275.81,E2 29275.81} C_VEL
LIN {X 0,Y 624.943,Z 977.845,A -85,B 0,C 180,E1 29274.218,E2 29274.218} C_VEL
LIN {X 0,Y 623.319,Z 995.485,A -85,B 0,C 180,E1 29272.723,E2 29272.723} C_VEL
LIN {X 0,Y 621.614,Z 1014.1,A -85,B 0,C 180,E1 29270.922,E2 29270.922} C_VEL
LIN {X 0,Y 620.349,Z 1028.931,A -85,B 0,C 180,E1 29269.295,E2 29269.295} C_VEL
LIN {X 0,Y 619.064,Z 1045.004,A -85,B 0,C 180,E1 29267.289,E2 29267.289} C_VEL
LIN {X 0,Y 618.158,Z 1057.613,A -85,B 0,C 180,E1 29265.48,E2 29265.48} C_VEL
LIN {X 0,Y 617.369,Z 1070.367,A -85,B 0,C 180,E1 29263.392,E2 29263.392} C_VEL
LIN {X 0,Y 616.777,Z 1081.119,A -85,B 0,C 180,E1 29261.313,E2 29261.313} C_VEL
LIN {X 0,Y 616.37,Z 1090.7,A -85,B 0,C 180,E1 29259.148,E2 29259.148} C_VEL
LIN {X 0,Y 616.114,Z 1098.092,A -85,B 0,C 180,E1 29257.085,E2 29257.085} C_VEL
LIN {X 0,Y 616.005,Z 1103.868,A -85,B 0,C 180,E1 29255.122,E2 29255.122} C_VEL
LIN {X 0,Y 615.933,Z 1109.072,A -85,B 0,C 180,E1 29252.791,E2 29252.791} C_VEL
LIN {X 0,Y 615.89,Z 1112.041,A -85,B 0,C 180,E1 29250.837,E2 29250.837} C_VEL
LIN {X 0,Y 615.893,Z 1113.785,A -85,B 0,C 180,E1 29248.977,E2 29248.977} C_VEL
LIN {X 0,Y 615.894,Z 1114.433,A -85,B 0,C 180,E1 29246.649,E2 29246.649} C_VEL
LIN {X 0,Y 615.909,Z 1113.54,A -85,B 0,C 180,E1 29244.597,E2 29244.597} C_VEL
LIN {X 0,Y 615.903,Z 1111.391,A -85,B 0,C 180,E1 29242.538,E2 29242.538} C_VEL
LIN {X 0,Y 615.934,Z 1107.391,A -85,B 0,C 180,E1 29240.28,E2 29240.28} C_VEL
LIN {X 0,Y 616.011,Z 1102.786,A -85,B 0,C 180,E1 29238.389,E2 29238.389} C_VEL
LIN {X 0,Y 616.201,Z 1096.073,A -85,B 0,C 180,E1 29236.2,E2 29236.2} C_VEL
LIN {X 0,Y 616.496,Z 1087.447,A -85,B 0,C 180,E1 29233.995,E2 29233.995} C_VEL
LIN {X 0,Y 616.926,Z 1078.083,A -85,B 0,C 180,E1 29231.967,E2 29231.967} C_VEL
LIN {X 0,Y 617.584,Z 1066.316,A -85,B 0,C 180,E1 29229.827,E2 29229.827} C_VEL
LIN {X 0,Y 618.405,Z 1054.07,A -85,B 0,C 180,E1 29227.893,E2 29227.893} C_VEL
LIN {X 0,Y 619.51,Z 1039.464,A -85,B 0,C 180,E1 29225.899,E2 29225.899} C_VEL
LIN {X 0,Y 620.635,Z 1025.451,A -85,B 0,C 180,E1 29224.215,E2 29224.215} C_VEL
LIN {X 0,Y 622.228,Z 1007.318,A -85,B 0,C 180,E1 29222.305,E2 29222.305} C_VEL
LIN {X 0,Y 623.912,Z 988.805,A -85,B 0,C 180,E1 29220.597,E2 29220.597} C_VEL
LIN {X 0,Y 625.758,Z 969.35,A -85,B 0,C 180,E1 29219.034,E2 29219.034} C_VEL
LIN {X 0,Y 627.361,Z 952.022,A -85,B 0,C 180,E1 29217.813,E2 29217.813} C_VEL
LIN {X 0,Y 629.28,Z 930.411,A -85,B 0,C 180,E1 29216.485,E2 29216.485} C_VEL
LIN {X 0,Y 630.932,Z 910.327,A -85,B 0,C 180,E1 29215.434,E2 29215.434} C_VEL
LIN {X 0,Y 632.659,Z 888.046,A -85,B 0,C 180,E1 29214.436,E2 29214.436} C_VEL
LIN {X 0,Y 634.118,Z 865.39,A -85,B 0,C 180,E1 29213.61,E2 29213.61} C_VEL
LIN {X 0,Y 635.373,Z 843.032,A -85,B 0,C 180,E1 29212.941,E2 29212.941} C_VEL
LIN {X 0,Y 636.424,Z 818.627,A -85,B 0,C 180,E1 29212.394,E2 29212.394} C_VEL
LIN {X 0,Y 637.119,Z 795.886,A -85,B 0,C 180,E1 29212.025,E2 29212.025} C_VEL
LIN {X 0,Y 641.269,Z 542.493,A -85,B 0,C 180,E1 29208.804,E2 29208.804} C_VEL
LIN {X 0,Y 642.598,Z 457.456,A -85,B 0,C 180,E1 29207.692,E2 29207.692} C_VEL
LIN {X 0,Y 632.422,Z 440.376,A -85,B 0,C 180,E1 29206.659,E2 29206.659} C_VEL
LIN {X 0,Y 622.163,Z 424.394,A -85,B 0,C 180,E1 29205.575,E2 29205.575} C_VEL
LIN {X 0,Y 617.365,Z 416.972,A -85,B 0,C 180,E1 29205.021,E2 29205.021} C_VEL
LIN {X 0,Y 616.988,Z 415.495,A -85,B 0,C 180,E1 29204.779,E2 29204.779} C_VEL
LIN {X 0,Y 616.917,Z 415.332,A -85,B 0,C 180,E1 29201.895,E2 29201.895} C_VEL
LIN {X 0,Y 617.005,Z 415.375,A -85,B 0,C 180,E1 29198.841,E2 29198.841} C_VEL
LIN {X 0,Y 616.925,Z 415.325,A -85,B 0,C 180,E1 29195.81,E2 29195.81} C_VEL
LIN {X 0,Y 617.007,Z 415.373,A -85,B 0,C 180,E1 29192.747,E2 29192.747} C_VEL
LIN {X 0,Y 616.936,Z 415.321,A -85,B 0,C 180,E1 29189.732,E2 29189.732} C_VEL
LIN {X 0,Y 617.013,Z 415.372,A -85,B 0,C 180,E1 29186.673,E2 29186.673} C_VEL
LIN {X 0,Y 616.949,Z 415.365,A -85,B 0,C 180,E1 29183.695,E2 29183.695} C_VEL
LIN {X 0,Y 617.017,Z 415.358,A -85,B 0,C 180,E1 29180.688,E2 29180.688} C_VEL
LIN {X 0,Y 616.958,Z 415.377,A -85,B 0,C 180,E1 29177.642,E2 29177.642} C_VEL
LIN {X 0,Y 617.018,Z 415.37,A -85,B 0,C 180,E1 29174.547,E2 29174.547} C_VEL
LIN {X 0,Y 616.964,Z 415.362,A -85,B 0,C 180,E1 29171.499,E2 29171.499} C_VEL
LIN {X 0,Y 617.015,Z 415.367,A -85,B 0,C 180,E1 29168.386,E2 29168.386} C_VEL
LIN {X 0,Y 616.975,Z 415.369,A -85,B 0,C 180,E1 29165.3,E2 29165.3} C_VEL
LIN {X 0,Y 617.01,Z 415.351,A -85,B 0,C 180,E1 29162.136,E2 29162.136} C_VEL
LIN {X 0,Y 616.992,Z 415.375,A -85,B 0,C 180,E1 29158.979,E2 29158.979} C_VEL
LIN {X 0,Y 617,Z 415.365,A -85,B 0,C 180,E1 29155.725,E2 29155.725} C_VEL
LIN {X 0,Y 617.012,Z 415.356,A -85,B 0,C 180,E1 29152.551,E2 29152.551} C_VEL
LIN {X 0,Y 616.993,Z 415.371,A -85,B 0,C 180,E1 29149.354,E2 29149.354} C_VEL
LIN {X 0,Y 617.001,Z 415.375,A -85,B 0,C 180,E1 29146.218,E2 29146.218} C_VEL
LIN {X 0,Y 616.994,Z 415.358,A -85,B 0,C 180,E1 29143.137,E2 29143.137} C_VEL
LIN {X 0,Y 616.996,Z 415.366,A -85,B 0,C 180,E1 29140.005,E2 29140.005} C_VEL
LIN {X 0,Y 617.002,Z 415.361,A -85,B 0,C 180,E1 29136.91,E2 29136.91} C_VEL
LIN {X 0,Y 616.991,Z 415.353,A -85,B 0,C 180,E1 29133.845,E2 29133.845} C_VEL
LIN {X 0,Y 617.013,Z 415.377,A -85,B 0,C 180,E1 29130.675,E2 29130.675} C_VEL
LIN {X 0,Y 617.001,Z 415.368,A -85,B 0,C 180,E1 29127.45,E2 29127.45} C_VEL
LIN {X 0,Y 616.991,Z 415.358,A -85,B 0,C 180,E1 29124.194,E2 29124.194} C_VEL
LIN {X 0,Y 617.017,Z 415.355,A -85,B 0,C 180,E1 29121.041,E2 29121.041} C_VEL
LIN {X 0,Y 616.974,Z 415.359,A -85,B 0,C 180,E1 29117.86,E2 29117.86} C_VEL
LIN {X 0,Y 617.033,Z 415.581,A -85,B 0,C 180,E1 29115.085,E2 29115.085} C_VEL
LIN {X 0,Y 624.496,Z 433.951,A -85,B 0,C 180,E1 29112.7,E2 29112.7} C_VEL
LIN {X 0,Y 630.663,Z 450.064,A -85,B 0,C 180,E1 29110.812,E2 29110.812} C_VEL
LIN {X 0,Y 637.328,Z 461.856,A -85,B 0,C 180,E1 29110.099,E2 29110.099} C_VEL
LIN {X 0,Y 642.585,Z 486.048,A -85,B 0,C 180,E1 29109.356,E2 29109.356} C_VEL
LIN {X 0,Y 638.608,Z 726.24,A -85,B 0,C 180,E1 29106.286,E2 29106.286} C_VEL
LIN {X 0,Y 636.717,Z 842.42,A -85,B 0,C 180,E1 29104.805,E2 29104.805} C_VEL
LIN {X 0,Y 635.741,Z 867.983,A -85,B 0,C 180,E1 29104.323,E2 29104.323} C_VEL
LIN {X 0,Y 634.708,Z 888.155,A -85,B 0,C 180,E1 29103.814,E2 29103.814} C_VEL
LIN {X 0,Y 633.374,Z 911.444,A -85,B 0,C 180,E1 29103.081,E2 29103.081} C_VEL
LIN {X 0,Y 631.752,Z 933.9,A -85,B 0,C 180,E1 29102.2,E2 29102.2} C_VEL
LIN {X 0,Y 630.142,Z 955.784,A -85,B 0,C 180,E1 29101.185,E2 29101.185} C_VEL
LIN {X 0,Y 628.335,Z 977.649,A -85,B 0,C 180,E1 29099.979,E2 29099.979} C_VEL
LIN {X 0,Y 626.737,Z 996.25,A -85,B 0,C 180,E1 29098.804,E2 29098.804} C_VEL
LIN {X 0,Y 624.83,Z 1017.764,A -85,B 0,C 180,E1 29097.237,E2 29097.237} C_VEL
LIN {X 0,Y 623.35,Z 1034.813,A -85,B 0,C 180,E1 29095.817,E2 29095.817} C_VEL
LIN {X 0,Y 621.654,Z 1053.67,A -85,B 0,C 180,E1 29094.013,E2 29094.013} C_VEL
LIN {X 0,Y 620.37,Z 1068.776,A -85,B 0,C 180,E1 29092.357,E2 29092.357} C_VEL
LIN {X 0,Y 619.12,Z 1084.411,A -85,B 0,C 180,E1 29090.417,E2 29090.417} C_VEL
LIN {X 0,Y 618.135,Z 1097.876,A -85,B 0,C 180,E1 29088.485,E2 29088.485} C_VEL
LIN {X 0,Y 617.334,Z 1110.733,A -85,B 0,C 180,E1 29086.369,E2 29086.369} C_VEL
LIN {X 0,Y 616.779,Z 1121.099,A -85,B 0,C 180,E1 29084.361,E2 29084.361} C_VEL
LIN {X 0,Y 616.376,Z 1130.771,A -85,B 0,C 180,E1 29082.174,E2 29082.174} C_VEL
LIN {X 0,Y 616.12,Z 1138.21,A -85,B 0,C 180,E1 29080.095,E2 29080.095} C_VEL
LIN {X 0,Y 616,Z 1143.999,A -85,B 0,C 180,E1 29078.118,E2 29078.118} C_VEL
LIN {X 0,Y 615.931,Z 1149.175,A -85,B 0,C 180,E1 29075.777,E2 29075.777} C_VEL
LIN {X 0,Y 615.915,Z 1152.123,A -85,B 0,C 180,E1 29073.816,E2 29073.816} C_VEL
LIN {X 0,Y 615.898,Z 1154.103,A -85,B 0,C 180,E1 29071.582,E2 29071.582} C_VEL
LIN {X 0,Y 615.884,Z 1154.372,A -85,B 0,C 180,E1 29069.442,E2 29069.442} C_VEL
LIN {X 0,Y 615.897,Z 1153.427,A -85,B 0,C 180,E1 29067.488,E2 29067.488} C_VEL
LIN {X 0,Y 615.908,Z 1150.769,A -85,B 0,C 180,E1 29065.157,E2 29065.157} C_VEL
LIN {X 0,Y 615.963,Z 1146.895,A -85,B 0,C 180,E1 29063.101,E2 29063.101} C_VEL
LIN {X 0,Y 616.033,Z 1141.71,A -85,B 0,C 180,E1 29061.036,E2 29061.036} C_VEL
LIN {X 0,Y 616.228,Z 1134.307,A -85,B 0,C 180,E1 29058.772,E2 29058.772} C_VEL
LIN {X 0,Y 616.528,Z 1126.749,A -85,B 0,C 180,E1 29056.876,E2 29056.876} C_VEL
LIN {X 0,Y 617.042,Z 1116.046,A -85,B 0,C 180,E1 29054.618,E2 29054.618} C_VEL
LIN {X 0,Y 617.67,Z 1105.114,A -85,B 0,C 180,E1 29052.671,E2 29052.671} C_VEL
LIN {X 0,Y 618.547,Z 1092.118,A -85,B 0,C 180,E1 29050.647,E2 29050.647} C_VEL
LIN {X 0,Y 619.639,Z 1077.613,A -85,B 0,C 180,E1 29048.711,E2 29048.711} C_VEL
LIN {X 0,Y 620.977,Z 1061.782,A -85,B 0,C 180,E1 29046.842,E2 29046.842} C_VEL
LIN {X 0,Y 622.442,Z 1044.821,A -85,B 0,C 180,E1 29045.11,E2 29045.11} C_VEL
LIN {X 0,Y 623.823,Z 1029.196,A -85,B 0,C 180,E1 29043.693,E2 29043.693} C_VEL
LIN {X 0,Y 625.643,Z 1008.741,A -85,B 0,C 180,E1 29042.078,E2 29042.078} C_VEL
LIN {X 0,Y 627.189,Z 991.068,A -85,B 0,C 180,E1 29040.854,E2 29040.854} C_VEL
LIN {X 0,Y 629.039,Z 969.239,A -85,B 0,C 180,E1 29039.531,E2 29039.531} C_VEL
LIN {X 0,Y 630.627,Z 949.36,A -85,B 0,C 180,E1 29038.502,E2 29038.502} C_VEL
LIN {X 0,Y 632.284,Z 927.536,A -85,B 0,C 180,E1 29037.528,E2 29037.528} C_VEL
LIN {X 0,Y 633.782,Z 904.117,A -85,B 0,C 180,E1 29036.673,E2 29036.673} C_VEL
LIN {X 0,Y 635.008,Z 882.596,A -85,B 0,C 180,E1 29036.029,E2 29036.029} C_VEL
LIN {X 0,Y 636.202,Z 857.149,A -85,B 0,C 180,E1 29035.451,E2 29035.451} C_VEL
LIN {X 0,Y 636.917,Z 835.053,A -85,B 0,C 180,E1 29035.089,E2 29035.089} C_VEL
LIN {X 0,Y 640.604,Z 597.743,A -85,B 0,C 180,E1 29032.083,E2 29032.083} C_VEL
LIN {X 0,Y 642.298,Z 484.465,A -85,B 0,C 180,E1 29030.626,E2 29030.626} C_VEL
LIN {X 0,Y 636.638,Z 460.626,A -85,B 0,C 180,E1 29029.878,E2 29029.878} C_VEL
LIN {X 0,Y 630.412,Z 449.852,A -85,B 0,C 180,E1 29029.232,E2 29029.232} C_VEL
LIN {X 0,Y 622.371,Z 428.964,A -85,B 0,C 180,E1 29026.835,E2 29026.835} C_VEL
LIN {X 0,Y 617.041,Z 415.555,A -85,B 0,C 180,E1 29025.158,E2 29025.158} C_VEL
LIN {X 0,Y 616.97,Z 415.312,A -85,B 0,C 180,E1 29022.076,E2 29022.076} C_VEL
LIN {X 0,Y 617.016,Z 415.373,A -85,B 0,C 180,E1 29018.84,E2 29018.84} C_VEL
LIN {X 0,Y 617.006,Z 415.368,A -85,B 0,C 180,E1 29015.576,E2 29015.576} C_VEL
LIN {X 0,Y 616.988,Z 415.362,A -85,B 0,C 180,E1 29012.33,E2 29012.33} C_VEL
LIN {X 0,Y 617.009,Z 415.356,A -85,B 0,C 180,E1 29009.302,E2 29009.302} C_VEL
LIN {X 0,Y 616.993,Z 415.374,A -85,B 0,C 180,E1 29006.128,E2 29006.128} C_VEL
LIN {X 0,Y 617.002,Z 415.365,A -85,B 0,C 180,E1 29002.989,E2 29002.989} C_VEL
LIN {X 0,Y 616.994,Z 415.364,A -85,B 0,C 180,E1 28999.897,E2 28999.897} C_VEL
LIN {X 0,Y 616.999,Z 415.372,A -85,B 0,C 180,E1 28996.766,E2 28996.766} C_VEL
LIN {X 0,Y 617.005,Z 415.354,A -85,B 0,C 180,E1 28993.591,E2 28993.591} C_VEL
LIN {X 0,Y 617.005,Z 415.366,A -85,B 0,C 180,E1 28990.363,E2 28990.363} C_VEL
LIN {X 0,Y 616.997,Z 415.37,A -85,B 0,C 180,E1 28987.075,E2 28987.075} C_VEL
LIN {X 0,Y 617.009,Z 415.36,A -85,B 0,C 180,E1 28983.903,E2 28983.903} C_VEL
LIN {X 0,Y 616.982,Z 415.375,A -85,B 0,C 180,E1 28980.743,E2 28980.743} C_VEL
LIN {X 0,Y 617.009,Z 415.353,A -85,B 0,C 180,E1 28977.678,E2 28977.678} C_VEL
LIN {X 0,Y 616.975,Z 415.374,A -85,B 0,C 180,E1 28974.606,E2 28974.606} C_VEL
LIN {X 0,Y 617.012,Z 415.35,A -85,B 0,C 180,E1 28971.52,E2 28971.52} C_VEL
LIN {X 0,Y 616.968,Z 415.372,A -85,B 0,C 180,E1 28968.407,E2 28968.407} C_VEL
LIN {X 0,Y 617.017,Z 415.357,A -85,B 0,C 180,E1 28965.261,E2 28965.261} C_VEL
LIN {X 0,Y 616.961,Z 415.367,A -85,B 0,C 180,E1 28962.261,E2 28962.261} C_VEL
LIN {X 0,Y 617.013,Z 415.37,A -85,B 0,C 180,E1 28959.113,E2 28959.113} C_VEL
LIN {X 0,Y 616.95,Z 415.355,A -85,B 0,C 180,E1 28956.199,E2 28956.199} C_VEL
LIN {X 0,Y 617.013,Z 415.372,A -85,B 0,C 180,E1 28953.119,E2 28953.119} C_VEL
LIN {X 0,Y 616.944,Z 415.375,A -85,B 0,C 180,E1 28950.161,E2 28950.161} C_VEL
LIN {X 0,Y 617.012,Z 415.358,A -85,B 0,C 180,E1 28947.12,E2 28947.12} C_VEL
LIN {X 0,Y 616.935,Z 415.374,A -85,B 0,C 180,E1 28944.076,E2 28944.076} C_VEL
LIN {X 0,Y 617.021,Z 415.374,A -85,B 0,C 180,E1 28941.041,E2 28941.041} C_VEL
LIN {X 0,Y 616.919,Z 415.32,A -85,B 0,C 180,E1 28938.068,E2 28938.068} C_VEL
LIN {X 0,Y 616.989,Z 415.375,A -85,B 0,C 180,E1 28935.089,E2 28935.089} C_VEL
LIN {X 0,Y 616.911,Z 415.324,A -85,B 0,C 180,E1 28932.02,E2 28932.02} C_VEL
LIN {X 0,Y 616.951,Z 415.377,A -85,B 0,C 180,E1 28929.203,E2 28929.203} C_VEL
LIN {X 0,Y 617.062,Z 415.773,A -85,B 0,C 180,E1 28928.867,E2 28928.867} C_VEL
LIN {X 0,Y 617.612,Z 417.641,A -85,B 0,C 180,E1 28928.675,E2 28928.675} C_VEL
LIN {X 0,Y 630.482,Z 437.702,A -85,B 0,C 180,E1 28927.369,E2 28927.369} C_VEL
LIN {X 0,Y 632.365,Z 440.676,A -85,B 0,C 180,E1 28927.183,E2 28927.183} C_VEL
LIN {X 0,Y 634.538,Z 445.074,A -85,B 0,C 180,E1 28926.955,E2 28926.955} C_VEL
LIN {X 0,Y 636.127,Z 452.292,A -85,B 0,C 180,E1 28926.733,E2 28926.733} C_VEL
LIN {X 0,Y 636.48,Z 462.44,A -85,B 0,C 180,E1 28926.562,E2 28926.562} C_VEL
LIN {X 0,Y 636.079,Z 475.211,A -85,B 0,C 180,E1 28926.409,E2 28926.409} C_VEL
LIN {X 0,Y 631.774,Z 726.346,A -85,B 0,C 180,E1 28923.191,E2 28923.191} C_VEL
LIN {X 0,Y 630.319,Z 806.177,A -85,B 0,C 180,E1 28922.154,E2 28922.154} C_VEL
LIN {X 0,Y 629.337,Z 831.198,A -85,B 0,C 180,E1 28921.668,E2 28921.668} C_VEL
LIN {X 0,Y 628.285,Z 851.171,A -85,B 0,C 180,E1 28921.153,E2 28921.153} C_VEL
LIN {X 0,Y 626.913,Z 873.872,A -85,B 0,C 180,E1 28920.424,E2 28920.424} C_VEL
LIN {X 0,Y 625.151,Z 896.608,A -85,B 0,C 180,E1 28919.514,E2 28919.514} C_VEL
LIN {X 0,Y 623.373,Z 918.907,A -85,B 0,C 180,E1 28918.45,E2 28918.45} C_VEL
LIN {X 0,Y 621.497,Z 939.28,A -85,B 0,C 180,E1 28917.292,E2 28917.292} C_VEL
LIN {X 0,Y 619.691,Z 958.155,A -85,B 0,C 180,E1 28916.065,E2 28916.065} C_VEL
LIN {X 0,Y 617.617,Z 978.754,A -85,B 0,C 180,E1 28914.515,E2 28914.515} C_VEL
LIN {X 0,Y 615.965,Z 995.419,A -85,B 0,C 180,E1 28913.081,E2 28913.081} C_VEL
LIN {X 0,Y 614.14,Z 1013.682,A -85,B 0,C 180,E1 28911.289,E2 28911.289} C_VEL
LIN {X 0,Y 612.55,Z 1030.956,A -85,B 0,C 180,E1 28909.352,E2 28909.352} C_VEL
LIN {X 0,Y 611.245,Z 1045.997,A -85,B 0,C 180,E1 28907.419,E2 28907.419} C_VEL
LIN {X 0,Y 610.289,Z 1058.513,A -85,B 0,C 180,E1 28905.587,E2 28905.587} C_VEL
LIN {X 0,Y 609.381,Z 1072.12,A -85,B 0,C 180,E1 28903.28,E2 28903.28} C_VEL
LIN {X 0,Y 608.819,Z 1081.906,A -85,B 0,C 180,E1 28901.338,E2 28901.338} C_VEL
LIN {X 0,Y 608.371,Z 1091.907,A -85,B 0,C 180,E1 28898.983,E2 28898.983} C_VEL
LIN {X 0,Y 608.115,Z 1098.824,A -85,B 0,C 180,E1 28896.989,E2 28896.989} C_VEL
LIN {X 0,Y 607.988,Z 1104.988,A -85,B 0,C 180,E1 28894.811,E2 28894.811} C_VEL
LIN {X 0,Y 607.932,Z 1109.616,A -85,B 0,C 180,E1 28892.545,E2 28892.545} C_VEL
LIN {X 0,Y 607.906,Z 1112.428,A -85,B 0,C 180,E1 28890.565,E2 28890.565} C_VEL
LIN {X 0,Y 607.901,Z 1114.206,A -85,B 0,C 180,E1 28888.209,E2 28888.209} C_VEL
LIN {X 0,Y 607.894,Z 1114.333,A -85,B 0,C 180,E1 28886.228,E2 28886.228} C_VEL
LIN {X 0,Y 607.907,Z 1113.238,A -85,B 0,C 180,E1 28884.147,E2 28884.147} C_VEL
LIN {X 0,Y 607.932,Z 1110.307,A -85,B 0,C 180,E1 28881.773,E2 28881.773} C_VEL
LIN {X 0,Y 607.976,Z 1106.468,A -85,B 0,C 180,E1 28879.769,E2 28879.769} C_VEL
LIN {X 0,Y 608.093,Z 1100.552,A -85,B 0,C 180,E1 28877.464,E2 28877.464} C_VEL
LIN {X 0,Y 608.313,Z 1093.419,A -85,B 0,C 180,E1 28875.337,E2 28875.337} C_VEL
LIN {X 0,Y 608.684,Z 1084.8,A -85,B 0,C 180,E1 28873.195,E2 28873.195} C_VEL
LIN {X 0,Y 609.236,Z 1074.285,A -85,B 0,C 180,E1 28871.037,E2 28871.037} C_VEL
LIN {X 0,Y 609.963,Z 1063.144,A -85,B 0,C 180,E1 28869.062,E2 28869.062} C_VEL
LIN {X 0,Y 610.987,Z 1049.462,A -85,B 0,C 180,E1 28866.975,E2 28866.975} C_VEL
LIN {X 0,Y 612.029,Z 1036.758,A -85,B 0,C 180,E1 28865.277,E2 28865.277} C_VEL
LIN {X 0,Y 613.593,Z 1019.614,A -85,B 0,C 180,E1 28863.254,E2 28863.254} C_VEL
LIN {X 0,Y 615.221,Z 1002.671,A -85,B 0,C 180,E1 28861.509,E2 28861.509} C_VEL
LIN {X 0,Y 617.216,Z 983.052,A -85,B 0,C 180,E1 28859.747,E2 28859.747} C_VEL
LIN {X 0,Y 618.873,Z 966.35,A -85,B 0,C 180,E1 28858.434,E2 28858.434} C_VEL
LIN {X 0,Y 620.887,Z 945.898,A -85,B 0,C 180,E1 28857.021,E2 28857.021} C_VEL
LIN {X 0,Y 622.701,Z 926.251,A -85,B 0,C 180,E1 28855.861,E2 28855.861} C_VEL
LIN {X 0,Y 624.493,Z 905.638,A -85,B 0,C 180,E1 28854.802,E2 28854.802} C_VEL
LIN {X 0,Y 626.247,Z 882.621,A -85,B 0,C 180,E1 28853.817,E2 28853.817} C_VEL
LIN {X 0,Y 627.675,Z 861.358,A -85,B 0,C 180,E1 28853.061,E2 28853.061} C_VEL
LIN {X 0,Y 629.068,Z 836.584,A -85,B 0,C 180,E1 28852.366,E2 28852.366} C_VEL
LIN {X 0,Y 630.007,Z 815.329,A -85,B 0,C 180,E1 28851.914,E2 28851.914} C_VEL
LIN {X 0,Y 630.772,Z 786.14,A -85,B 0,C 180,E1 28851.477,E2 28851.477} C_VEL
LIN {X 0,Y 635.148,Z 537.396,A -85,B 0,C 180,E1 28848.283,E2 28848.283} C_VEL
LIN {X 0,Y 636.489,Z 460.71,A -85,B 0,C 180,E1 28847.275,E2 28847.275} C_VEL
LIN {X 0,Y 625.113,Z 441.75,A -85,B 0,C 180,E1 28846.087,E2 28846.087} C_VEL
LIN {X 0,Y 614.628,Z 425.748,A -85,B 0,C 180,E1 28844.947,E2 28844.947} C_VEL
LIN {X 0,Y 611.563,Z 421.305,A -85,B 0,C 180,E1 28844.606,E2 28844.606} C_VEL
LIN {X 0,Y 609.428,Z 418.162,A -85,B 0,C 180,E1 28844.359,E2 28844.359} C_VEL
LIN {X 0,Y 609.019,Z 416.626,A -85,B 0,C 180,E1 28844.176,E2 28844.176} C_VEL
LIN {X 0,Y 608.988,Z 416.316,A -85,B 0,C 180,E1 28841.663,E2 28841.663} C_VEL
LIN {X 0,Y 609.006,Z 416.365,A -85,B 0,C 180,E1 28838.361,E2 28838.361} C_VEL
LIN {X 0,Y 608.999,Z 416.313,A -85,B 0,C 180,E1 28835.536,E2 28835.536} C_VEL
LIN {X 0,Y 609.014,Z 416.363,A -85,B 0,C 180,E1 28832.249,E2 28832.249} C_VEL
LIN {X 0,Y 609.005,Z 416.306,A -85,B 0,C 180,E1 28829.509,E2 28829.509} C_VEL
LIN {X 0,Y 609.038,Z 416.366,A -85,B 0,C 180,E1 28826.311,E2 28826.311} C_VEL
LIN {X 0,Y 609.02,Z 416.355,A -85,B 0,C 180,E1 28823.398,E2 28823.398} C_VEL
LIN {X 0,Y 609.033,Z 416.348,A -85,B 0,C 180,E1 28820.1,E2 28820.1} C_VEL
LIN {X 0,Y 609.046,Z 416.361,A -85,B 0,C 180,E1 28817.09,E2 28817.09} C_VEL
LIN {X 0,Y 609.034,Z 416.363,A -85,B 0,C 180,E1 28813.869,E2 28813.869} C_VEL
LIN {X 0,Y 609.068,Z 416.348,A -85,B 0,C 180,E1 28810.787,E2 28810.787} C_VEL
LIN {X 0,Y 609.033,Z 416.357,A -85,B 0,C 180,E1 28807.642,E2 28807.642} C_VEL
LIN {X 0,Y 609.075,Z 416.363,A -85,B 0,C 180,E1 28804.52,E2 28804.52} C_VEL
LIN {X 0,Y 609.037,Z 416.345,A -85,B 0,C 180,E1 28801.317,E2 28801.317} C_VEL
LIN {X 0,Y 609.07,Z 416.346,A -85,B 0,C 180,E1 28798.213,E2 28798.213} C_VEL
LIN {X 0,Y 609.053,Z 416.36,A -85,B 0,C 180,E1 28795.008,E2 28795.008} C_VEL
LIN {X 0,Y 609.066,Z 416.349,A -85,B 0,C 180,E1 28791.694,E2 28791.694} C_VEL
LIN {X 0,Y 609.067,Z 416.346,A -85,B 0,C 180,E1 28788.446,E2 28788.446} C_VEL
LIN {X 0,Y 609.056,Z 416.362,A -85,B 0,C 180,E1 28785.233,E2 28785.233} C_VEL
LIN {X 0,Y 609.06,Z 416.359,A -85,B 0,C 180,E1 28782.122,E2 28782.122} C_VEL
LIN {X 0,Y 609.06,Z 416.342,A -85,B 0,C 180,E1 28778.928,E2 28778.928} C_VEL
LIN {X 0,Y 609.06,Z 416.361,A -85,B 0,C 180,E1 28775.768,E2 28775.768} C_VEL
LIN {X 0,Y 609.07,Z 416.341,A -85,B 0,C 180,E1 28772.528,E2 28772.528} C_VEL
LIN {X 0,Y 609.076,Z 416.345,A -85,B 0,C 180,E1 28769.299,E2 28769.299} C_VEL
LIN {X 0,Y 609.049,Z 416.362,A -85,B 0,C 180,E1 28766.069,E2 28766.069} C_VEL
LIN {X 0,Y 609.075,Z 416.361,A -85,B 0,C 180,E1 28762.925,E2 28762.925} C_VEL
LIN {X 0,Y 609.037,Z 416.359,A -85,B 0,C 180,E1 28759.767,E2 28759.767} C_VEL
LIN {X 0,Y 609.075,Z 416.35,A -85,B 0,C 180,E1 28756.657,E2 28756.657} C_VEL
LIN {X 0,Y 609.073,Z 416.639,A -85,B 0,C 180,E1 28755.72,E2 28755.72} C_VEL
LIN {X 0,Y 616.815,Z 435.321,A -85,B 0,C 180,E1 28753.225,E2 28753.225} C_VEL
LIN {X 0,Y 622.482,Z 449.759,A -85,B 0,C 180,E1 28751.484,E2 28751.484} C_VEL
LIN {X 0,Y 631.791,Z 466.133,A -85,B 0,C 180,E1 28750.469,E2 28750.469} C_VEL
LIN {X 0,Y 636.388,Z 487.817,A -85,B 0,C 180,E1 28749.794,E2 28749.794} C_VEL
LIN {X 0,Y 632.131,Z 727.654,A -85,B 0,C 180,E1 28746.697,E2 28746.697} C_VEL
LIN {X 0,Y 630.127,Z 842.217,A -85,B 0,C 180,E1 28745.221,E2 28745.221} C_VEL
LIN {X 0,Y 629.082,Z 867.879,A -85,B 0,C 180,E1 28744.733,E2 28744.733} C_VEL
LIN {X 0,Y 627.975,Z 888.24,A -85,B 0,C 180,E1 28744.214,E2 28744.214} C_VEL
LIN {X 0,Y 626.527,Z 911.785,A -85,B 0,C 180,E1 28743.463,E2 28743.463} C_VEL
LIN {X 0,Y 624.831,Z 934.011,A -85,B 0,C 180,E1 28742.581,E2 28742.581} C_VEL
LIN {X 0,Y 623.088,Z 956.128,A -85,B 0,C 180,E1 28741.544,E2 28741.544} C_VEL
LIN {X 0,Y 621.212,Z 977.344,A -85,B 0,C 180,E1 28740.359,E2 28740.359} C_VEL
LIN {X 0,Y 619.516,Z 995.958,A -85,B 0,C 180,E1 28739.171,E2 28739.171} C_VEL
LIN {X 0,Y 617.468,Z 1017.459,A -85,B 0,C 180,E1 28737.589,E2 28737.589} C_VEL
LIN {X 0,Y 615.925,Z 1033.947,A -85,B 0,C 180,E1 28736.204,E2 28736.204} C_VEL
LIN {X 0,Y 614.198,Z 1052.655,A -85,B 0,C 180,E1 28734.425,E2 28734.425} C_VEL
LIN {X 0,Y 612.881,Z 1067.083,A -85,B 0,C 180,E1 28732.848,E2 28732.848} C_VEL
LIN {X 0,Y 611.585,Z 1082.234,A -85,B 0,C 180,E1 28730.98,E2 28730.98} C_VEL
LIN {X 0,Y 610.429,Z 1096.604,A -85,B 0,C 180,E1 28728.925,E2 28728.925} C_VEL
LIN {X 0,Y 609.565,Z 1109.121,A -85,B 0,C 180,E1 28726.878,E2 28726.878} C_VEL
LIN {X 0,Y 608.901,Z 1120.34,A -85,B 0,C 180,E1 28724.712,E2 28724.712} C_VEL
LIN {X 0,Y 608.482,Z 1129.178,A -85,B 0,C 180,E1 28722.721,E2 28722.721} C_VEL
LIN {X 0,Y 608.171,Z 1137.604,A -85,B 0,C 180,E1 28720.419,E2 28720.419} C_VEL
LIN {X 0,Y 608.026,Z 1143.49,A -85,B 0,C 180,E1 28718.416,E2 28718.416} C_VEL
LIN {X 0,Y 607.949,Z 1148.696,A -85,B 0,C 180,E1 28716.137,E2 28716.137} C_VEL
LIN {X 0,Y 607.918,Z 1152.009,A -85,B 0,C 180,E1 28713.961,E2 28713.961} C_VEL
LIN {X 0,Y 607.906,Z 1153.903,A -85,B 0,C 180,E1 28711.885,E2 28711.885} C_VEL
LIN {X 0,Y 607.884,Z 1154.395,A -85,B 0,C 180,E1 28709.529,E2 28709.529} C_VEL
LIN {X 0,Y 607.901,Z 1153.495,A -85,B 0,C 180,E1 28707.549,E2 28707.549} C_VEL
LIN {X 0,Y 607.916,Z 1151.085,A -85,B 0,C 180,E1 28705.283,E2 28705.283} C_VEL
LIN {X 0,Y 607.964,Z 1147.102,A -85,B 0,C 180,E1 28703.104,E2 28703.104} C_VEL
LIN {X 0,Y 608.033,Z 1142.219,A -85,B 0,C 180,E1 28701.108,E2 28701.108} C_VEL
LIN {X 0,Y 608.248,Z 1134.66,A -85,B 0,C 180,E1 28698.719,E2 28698.719} C_VEL
LIN {X 0,Y 608.58,Z 1126.748,A -85,B 0,C 180,E1 28696.702,E2 28696.702} C_VEL
LIN {X 0,Y 609.122,Z 1116.402,A -85,B 0,C 180,E1 28694.48,E2 28694.48} C_VEL
LIN {X 0,Y 609.829,Z 1105.112,A -85,B 0,C 180,E1 28692.441,E2 28692.441} C_VEL
LIN {X 0,Y 610.777,Z 1092.116,A -85,B 0,C 180,E1 28690.391,E2 28690.391} C_VEL
LIN {X 0,Y 611.884,Z 1078.381,A -85,B 0,C 180,E1 28688.528,E2 28688.528} C_VEL
LIN {X 0,Y 613.286,Z 1062.857,A -85,B 0,C 180,E1 28686.66,E2 28686.66} C_VEL
LIN {X 0,Y 614.837,Z 1045.658,A -85,B 0,C 180,E1 28684.884,E2 28684.884} C_VEL
LIN {X 0,Y 616.394,Z 1028.969,A -85,B 0,C 180,E1 28683.357,E2 28683.357} C_VEL
LIN {X 0,Y 618.341,Z 1008.448,A -85,B 0,C 180,E1 28681.719,E2 28681.719} C_VEL
LIN {X 0,Y 620.052,Z 990.032,A -85,B 0,C 180,E1 28680.432,E2 28680.432} C_VEL
LIN {X 0,Y 622.131,Z 967.133,A -85,B 0,C 180,E1 28679.049,E2 28679.049} C_VEL
LIN {X 0,Y 623.747,Z 948.083,A -85,B 0,C 180,E1 28678.062,E2 28678.062} C_VEL
LIN {X 0,Y 625.516,Z 926.062,A -85,B 0,C 180,E1 28677.078,E2 28677.078} C_VEL
LIN {X 0,Y 627.05,Z 903.081,A -85,B 0,C 180,E1 28676.24,E2 28676.24} C_VEL
LIN {X 0,Y 628.461,Z 879.973,A -85,B 0,C 180,E1 28675.552,E2 28675.552} C_VEL
LIN {X 0,Y 629.635,Z 855.842,A -85,B 0,C 180,E1 28675.017,E2 28675.017} C_VEL
LIN {X 0,Y 630.379,Z 833.466,A -85,B 0,C 180,E1 28674.652,E2 28674.652} C_VEL
LIN {X 0,Y 634.247,Z 596.949,A -85,B 0,C 180,E1 28671.634,E2 28671.634} C_VEL
LIN {X 0,Y 636.026,Z 486.275,A -85,B 0,C 180,E1 28670.198,E2 28670.198} C_VEL
LIN {X 0,Y 630.891,Z 464.723,A -85,B 0,C 180,E1 28669.513,E2 28669.513} C_VEL
LIN {X 0,Y 622.151,Z 449.613,A -85,B 0,C 180,E1 28668.603,E2 28668.603} C_VEL
LIN {X 0,Y 614.184,Z 429.46,A -85,B 0,C 180,E1 28666.219,E2 28666.219} C_VEL
LIN {X 0,Y 609.065,Z 416.545,A -85,B 0,C 180,E1 28664.562,E2 28664.562} C_VEL
LIN {X 0,Y 609.069,Z 416.291,A -85,B 0,C 180,E1 28661.53,E2 28661.53} C_VEL
LIN {X 0,Y 609.041,Z 416.367,A -85,B 0,C 180,E1 28658.302,E2 28658.302} C_VEL
LIN {X 0,Y 609.073,Z 416.367,A -85,B 0,C 180,E1 28655.16,E2 28655.16} C_VEL
LIN {X 0,Y 609.046,Z 416.353,A -85,B 0,C 180,E1 28652.025,E2 28652.025} C_VEL
LIN {X 0,Y 609.066,Z 416.341,A -85,B 0,C 180,E1 28648.953,E2 28648.953} C_VEL
LIN {X 0,Y 609.058,Z 416.364,A -85,B 0,C 180,E1 28645.789,E2 28645.789} C_VEL
LIN {X 0,Y 609.081,Z 416.354,A -85,B 0,C 180,E1 28642.489,E2 28642.489} C_VEL
LIN {X 0,Y 609.067,Z 416.344,A -85,B 0,C 180,E1 28639.267,E2 28639.267} C_VEL
LIN {X 0,Y 609.062,Z 416.361,A -85,B 0,C 180,E1 28636.01,E2 28636.01} C_VEL
LIN {X 0,Y 609.055,Z 416.356,A -85,B 0,C 180,E1 28632.901,E2 28632.901} C_VEL
LIN {X 0,Y 609.064,Z 416.352,A -85,B 0,C 180,E1 28629.735,E2 28629.735} C_VEL
LIN {X 0,Y 609.051,Z 416.361,A -85,B 0,C 180,E1 28626.599,E2 28626.599} C_VEL
LIN {X 0,Y 609.071,Z 416.341,A -85,B 0,C 180,E1 28623.388,E2 28623.388} C_VEL
LIN {X 0,Y 609.061,Z 416.359,A -85,B 0,C 180,E1 28620.188,E2 28620.188} C_VEL
LIN {X 0,Y 609.046,Z 416.347,A -85,B 0,C 180,E1 28616.894,E2 28616.894} C_VEL
LIN {X 0,Y 609.076,Z 416.359,A -85,B 0,C 180,E1 28613.78,E2 28613.78} C_VEL
LIN {X 0,Y 609.033,Z 416.358,A -85,B 0,C 180,E1 28610.646,E2 28610.646} C_VEL
LIN {X 0,Y 609.076,Z 416.351,A -85,B 0,C 180,E1 28607.485,E2 28607.485} C_VEL
LIN {X 0,Y 609.025,Z 416.364,A -85,B 0,C 180,E1 28604.38,E2 28604.38} C_VEL
LIN {X 0,Y 609.074,Z 416.342,A -85,B 0,C 180,E1 28601.23,E2 28601.23} C_VEL
LIN {X 0,Y 609.016,Z 416.364,A -85,B 0,C 180,E1 28598.219,E2 28598.219} C_VEL
LIN {X 0,Y 609.073,Z 416.344,A -85,B 0,C 180,E1 28595.149,E2 28595.149} C_VEL
LIN {X 0,Y 609.009,Z 416.355,A -85,B 0,C 180,E1 28592.1,E2 28592.1} C_VEL
LIN {X 0,Y 609.065,Z 416.364,A -85,B 0,C 180,E1 28588.97,E2 28588.97} C_VEL
LIN {X 0,Y 609.001,Z 416.364,A -85,B 0,C 180,E1 28585.953,E2 28585.953} C_VEL
LIN {X 0,Y 609.049,Z 416.352,A -85,B 0,C 180,E1 28582.832,E2 28582.832} C_VEL
LIN {X 0,Y 608.99,Z 416.359,A -85,B 0,C 180,E1 28580.06,E2 28580.06} C_VEL
LIN {X 0,Y 609.052,Z 416.303,A -85,B 0,C 180,E1 28577.053,E2 28577.053} C_VEL
LIN {X 0,Y 608.98,Z 416.359,A -85,B 0,C 180,E1 28573.99,E2 28573.99} C_VEL
LIN {X 0,Y 609.052,Z 416.311,A -85,B 0,C 180,E1 28570.923,E2 28570.923} C_VEL
LIN {X 0,Y 609.026,Z 416.66,A -85,B 0,C 180,E1 28569.498,E2 28569.498} C_VEL
LIN {X 0,Y 609.25,Z 417.616,A -85,B 0,C 180,E1 28569.376,E2 28569.376} C_VEL
LIN {X 0,Y 611.158,Z 420.892,A -85,B 0,C 180,E1 28569.15,E2 28569.15} C_VEL
LIN {X 0,Y 612.603,Z 422.824,A -85,B 0,C 180,E1 28569.001,E2 28569.001} C_VEL
LIN {X 0,Y 625.565,Z 443.127,A -85,B 0,C 180,E1 28567.664,E2 28567.664} C_VEL
LIN {X 0,Y 636.329,Z 460.834,A -85,B 0,C 180,E1 28566.596,E2 28566.596} C_VEL
LIN {X 0,Y 636.079,Z 475.211,A -85,B 0,C 180,E1 28566.409,E2 28566.409} C_VEL
LIN {X 0,Y 635.2,Z 482.906,A -85,B 0,C 180,E1 28566.364,E2 28566.364} C_VEL
LIN {X 0,Y 629.942,Z 503.474,A -85,B 0,C 180,E1 28566.457,E2 28566.457} C_VEL
LIN {X 0,Y 629.215,Z 510.082,A -85,B 0,C 180,E1 28566.416,E2 28566.416} C_VEL
LIN {X 0,Y 624.806,Z 754.648,A -85,B 0,C 180,E1 28563.263,E2 28563.263} C_VEL
LIN {X 0,Y 623.751,Z 808.383,A -85,B 0,C 180,E1 28562.547,E2 28562.547} C_VEL
LIN {X 0,Y 622.713,Z 832.418,A -85,B 0,C 180,E1 28562.065,E2 28562.065} C_VEL
LIN {X 0,Y 621.614,Z 852.245,A -85,B 0,C 180,E1 28561.546,E2 28561.546} C_VEL
LIN {X 0,Y 620.123,Z 875.223,A -85,B 0,C 180,E1 28560.793,E2 28560.793} C_VEL
LIN {X 0,Y 618.376,Z 896.723,A -85,B 0,C 180,E1 28559.923,E2 28559.923} C_VEL
LIN {X 0,Y 616.561,Z 918.094,A -85,B 0,C 180,E1 28558.9,E2 28558.9} C_VEL
LIN {X 0,Y 614.502,Z 939.45,A -85,B 0,C 180,E1 28557.681,E2 28557.681} C_VEL
LIN {X 0,Y 612.62,Z 958.075,A -85,B 0,C 180,E1 28556.46,E2 28556.46} C_VEL
LIN {X 0,Y 610.414,Z 978.714,A -85,B 0,C 180,E1 28554.897,E2 28554.897} C_VEL
LIN {X 0,Y 608.618,Z 995.633,A -85,B 0,C 180,E1 28553.427,E2 28553.427} C_VEL
LIN {X 0,Y 606.63,Z 1014.359,A -85,B 0,C 180,E1 28551.566,E2 28551.566} C_VEL
LIN {X 0,Y 605.131,Z 1029.003,A -85,B 0,C 180,E1 28549.9,E2 28549.9} C_VEL
LIN {X 0,Y 603.621,Z 1044.916,A -85,B 0,C 180,E1 28547.846,E2 28547.846} C_VEL
LIN {X 0,Y 602.568,Z 1057.531,A -85,B 0,C 180,E1 28545.989,E2 28545.989} C_VEL
LIN {X 0,Y 601.623,Z 1070.304,A -85,B 0,C 180,E1 28543.847,E2 28543.847} C_VEL
LIN {X 0,Y 600.959,Z 1080.604,A -85,B 0,C 180,E1 28541.809,E2 28541.809} C_VEL
LIN {X 0,Y 600.507,Z 1089.465,A -85,B 0,C 180,E1 28539.778,E2 28539.778} C_VEL
LIN {X 0,Y 600.186,Z 1097.749,A -85,B 0,C 180,E1 28537.466,E2 28537.466} C_VEL
LIN {X 0,Y 600.024,Z 1103.326,A -85,B 0,C 180,E1 28535.546,E2 28535.546} C_VEL
LIN {X 0,Y 599.925,Z 1108.571,A -85,B 0,C 180,E1 28533.249,E2 28533.249} C_VEL
LIN {X 0,Y 599.891,Z 1111.91,A -85,B 0,C 180,E1 28531.051,E2 28531.051} C_VEL
LIN {X 0,Y 599.902,Z 1113.706,A -85,B 0,C 180,E1 28529.14,E2 28529.14} C_VEL
LIN {X 0,Y 599.898,Z 1114.459,A -85,B 0,C 180,E1 28526.751,E2 28526.751} C_VEL
LIN {X 0,Y 599.907,Z 1113.618,A -85,B 0,C 180,E1 28524.644,E2 28524.644} C_VEL
LIN {X 0,Y 599.893,Z 1111.75,A -85,B 0,C 180,E1 28522.722,E2 28522.722} C_VEL
LIN {X 0,Y 599.93,Z 1108.045,A -85,B 0,C 180,E1 28520.406,E2 28520.406} C_VEL
LIN {X 0,Y 600.023,Z 1103.336,A -85,B 0,C 180,E1 28518.367,E2 28518.367} C_VEL
LIN {X 0,Y 600.19,Z 1097.66,A -85,B 0,C 180,E1 28516.414,E2 28516.414} C_VEL
LIN {X 0,Y 600.525,Z 1089.143,A -85,B 0,C 180,E1 28514.054,E2 28514.054} C_VEL
LIN {X 0,Y 600.966,Z 1080.474,A -85,B 0,C 180,E1 28512.073,E2 28512.073} C_VEL
LIN {X 0,Y 601.689,Z 1069.302,A -85,B 0,C 180,E1 28509.88,E2 28509.88} C_VEL
LIN {X 0,Y 602.625,Z 1056.74,A -85,B 0,C 180,E1 28507.797,E2 28507.797} C_VEL
LIN {X 0,Y 603.853,Z 1042.7,A -85,B 0,C 180,E1 28505.754,E2 28505.754} C_VEL
LIN {X 0,Y 605.28,Z 1027.489,A -85,B 0,C 180,E1 28503.828,E2 28503.828} C_VEL
LIN {X 0,Y 607.007,Z 1011.176,A -85,B 0,C 180,E1 28501.998,E2 28501.998} C_VEL
LIN {X 0,Y 608.856,Z 993.29,A -85,B 0,C 180,E1 28500.267,E2 28500.267} C_VEL
LIN {X 0,Y 610.881,Z 974.883,A -85,B 0,C 180,E1 28498.695,E2 28498.695} C_VEL
LIN {X 0,Y 612.899,Z 955.37,A -85,B 0,C 180,E1 28497.261,E2 28497.261} C_VEL
LIN {X 0,Y 614.817,Z 936.449,A -85,B 0,C 180,E1 28496.04,E2 28496.04} C_VEL
LIN {X 0,Y 616.894,Z 914.248,A -85,B 0,C 180,E1 28494.815,E2 28494.815} C_VEL
LIN {X 0,Y 618.554,Z 894.888,A -85,B 0,C 180,E1 28493.904,E2 28493.904} C_VEL
LIN {X 0,Y 620.435,Z 870.92,A -85,B 0,C 180,E1 28492.963,E2 28492.963} C_VEL
LIN {X 0,Y 621.767,Z 849.874,A -85,B 0,C 180,E1 28492.294,E2 28492.294} C_VEL
LIN {X 0,Y 622.951,Z 828.307,A -85,B 0,C 180,E1 28491.745,E2 28491.745} C_VEL
LIN {X 0,Y 623.88,Z 803.307,A -85,B 0,C 180,E1 28491.282,E2 28491.282} C_VEL
LIN {X 0,Y 628.397,Z 566.754,A -85,B 0,C 180,E1 28488.202,E2 28488.202} C_VEL
LIN {X 0,Y 630.337,Z 463.986,A -85,B 0,C 180,E1 28486.844,E2 28486.844} C_VEL
LIN {X 0,Y 619.976,Z 446.631,A -85,B 0,C 180,E1 28485.732,E2 28485.732} C_VEL
LIN {X 0,Y 609.963,Z 431.301,A -85,B 0,C 180,E1 28484.622,E2 28484.622} C_VEL
LIN {X 0,Y 607.072,Z 427.17,A -85,B 0,C 180,E1 28484.296,E2 28484.296} C_VEL
LIN {X 0,Y 603.893,Z 422.558,A -85,B 0,C 180,E1 28483.928,E2 28483.928} C_VEL
LIN {X 0,Y 601.674,Z 419.595,A -85,B 0,C 180,E1 28483.67,E2 28483.67} C_VEL
LIN {X 0,Y 601.132,Z 417.783,A -85,B 0,C 180,E1 28483.513,E2 28483.513} C_VEL
LIN {X 0,Y 601.113,Z 417.314,A -85,B 0,C 180,E1 28483,E2 28483} C_VEL
LIN {X 0,Y 601.046,Z 417.337,A -85,B 0,C 180,E1 28479.952,E2 28479.952} C_VEL
LIN {X 0,Y 601.116,Z 417.296,A -85,B 0,C 180,E1 28477.019,E2 28477.019} C_VEL
LIN {X 0,Y 601.058,Z 417.354,A -85,B 0,C 180,E1 28473.869,E2 28473.869} C_VEL
LIN {X 0,Y 601.136,Z 417.297,A -85,B 0,C 180,E1 28470.818,E2 28470.818} C_VEL
LIN {X 0,Y 601.066,Z 417.334,A -85,B 0,C 180,E1 28467.748,E2 28467.748} C_VEL
LIN {X 0,Y 601.137,Z 417.336,A -85,B 0,C 180,E1 28464.677,E2 28464.677} C_VEL
LIN {X 0,Y 601.076,Z 417.356,A -85,B 0,C 180,E1 28461.672,E2 28461.672} C_VEL
LIN {X 0,Y 601.138,Z 417.352,A -85,B 0,C 180,E1 28458.524,E2 28458.524} C_VEL
LIN {X 0,Y 601.083,Z 417.336,A -85,B 0,C 180,E1 28455.436,E2 28455.436} C_VEL
LIN {X 0,Y 601.13,Z 417.337,A -85,B 0,C 180,E1 28452.293,E2 28452.293} C_VEL
LIN {X 0,Y 601.101,Z 417.354,A -85,B 0,C 180,E1 28449.189,E2 28449.189} C_VEL
LIN {X 0,Y 601.113,Z 417.342,A -85,B 0,C 180,E1 28445.892,E2 28445.892} C_VEL
LIN {X 0,Y 601.127,Z 417.335,A -85,B 0,C 180,E1 28442.765,E2 28442.765} C_VEL
LIN {X 0,Y 601.105,Z 417.349,A -85,B 0,C 180,E1 28439.523,E2 28439.523} C_VEL
LIN {X 0,Y 601.129,Z 417.336,A -85,B 0,C 180,E1 28436.376,E2 28436.376} C_VEL
LIN {X 0,Y 601.107,Z 417.34,A -85,B 0,C 180,E1 28433.217,E2 28433.217} C_VEL
LIN {X 0,Y 601.13,Z 417.348,A -85,B 0,C 180,E1 28430.038,E2 28430.038} C_VEL
LIN {X 0,Y 601.129,Z 417.338,A -85,B 0,C 180,E1 28426.73,E2 28426.73} C_VEL
LIN {X 0,Y 601.129,Z 417.333,A -85,B 0,C 180,E1 28423.475,E2 28423.475} C_VEL
LIN {X 0,Y 601.122,Z 417.346,A -85,B 0,C 180,E1 28420.265,E2 28420.265} C_VEL
LIN {X 0,Y 601.124,Z 417.336,A -85,B 0,C 180,E1 28417.093,E2 28417.093} C_VEL
LIN {X 0,Y 601.114,Z 417.33,A -85,B 0,C 180,E1 28413.927,E2 28413.927} C_VEL
LIN {X 0,Y 601.135,Z 417.354,A -85,B 0,C 180,E1 28410.724,E2 28410.724} C_VEL
LIN {X 0,Y 601.121,Z 417.344,A -85,B 0,C 180,E1 28407.494,E2 28407.494} C_VEL
LIN {X 0,Y 601.113,Z 417.334,A -85,B 0,C 180,E1 28404.16,E2 28404.16} C_VEL
LIN {X 0,Y 601.136,Z 417.33,A -85,B 0,C 180,E1 28400.967,E2 28400.967} C_VEL
LIN {X 0,Y 601.097,Z 417.336,A -85,B 0,C 180,E1 28397.894,E2 28397.894} C_VEL
LIN {X 0,Y 601.157,Z 417.537,A -85,B 0,C 180,E1 28396.411,E2 28396.411} C_VEL
LIN {X 0,Y 603.963,Z 424.485,A -85,B 0,C 180,E1 28395.416,E2 28395.416} C_VEL
LIN {X 0,Y 611.552,Z 442.836,A -85,B 0,C 180,E1 28392.985,E2 28392.985} C_VEL
LIN {X 0,Y 614.214,Z 449.473,A -85,B 0,C 180,E1 28392.191,E2 28392.191} C_VEL
LIN {X 0,Y 626.171,Z 470.013,A -85,B 0,C 180,E1 28390.861,E2 28390.861} C_VEL
LIN {X 0,Y 630.258,Z 489.671,A -85,B 0,C 180,E1 28390.242,E2 28390.242} C_VEL
LIN {X 0,Y 625.722,Z 728.421,A -85,B 0,C 180,E1 28387.129,E2 28387.129} C_VEL
LIN {X 0,Y 623.587,Z 841.94,A -85,B 0,C 180,E1 28385.648,E2 28385.648} C_VEL
LIN {X 0,Y 622.468,Z 867.633,A -85,B 0,C 180,E1 28385.155,E2 28385.155} C_VEL
LIN {X 0,Y 621.27,Z 888.425,A -85,B 0,C 180,E1 28384.62,E2 28384.62} C_VEL
LIN {X 0,Y 619.761,Z 911.48,A -85,B 0,C 180,E1 28383.877,E2 28383.877} C_VEL
LIN {X 0,Y 617.976,Z 933.706,A -85,B 0,C 180,E1 28382.988,E2 28382.988} C_VEL
LIN {X 0,Y 616.193,Z 954.81,A -85,B 0,C 180,E1 28381.993,E2 28381.993} C_VEL
LIN {X 0,Y 614.116,Z 977.039,A -85,B 0,C 180,E1 28380.747,E2 28380.747} C_VEL
LIN {X 0,Y 612.318,Z 995.641,A -85,B 0,C 180,E1 28379.548,E2 28379.548} C_VEL
LIN {X 0,Y 610.137,Z 1017.154,A -85,B 0,C 180,E1 28377.95,E2 28377.95} C_VEL
LIN {X 0,Y 608.435,Z 1034.093,A -85,B 0,C 180,E1 28376.509,E2 28376.509} C_VEL
LIN {X 0,Y 606.516,Z 1053.569,A -85,B 0,C 180,E1 28374.62,E2 28374.62} C_VEL
LIN {X 0,Y 605.091,Z 1068.61,A -85,B 0,C 180,E1 28372.953,E2 28372.953} C_VEL
LIN {X 0,Y 603.751,Z 1083.706,A -85,B 0,C 180,E1 28371.062,E2 28371.062} C_VEL
LIN {X 0,Y 602.586,Z 1097.237,A -85,B 0,C 180,E1 28369.08,E2 28369.08} C_VEL
LIN {X 0,Y 601.671,Z 1109.688,A -85,B 0,C 180,E1 28367.007,E2 28367.007} C_VEL
LIN {X 0,Y 600.968,Z 1120.695,A -85,B 0,C 180,E1 28364.834,E2 28364.834} C_VEL
LIN {X 0,Y 600.5,Z 1129.988,A -85,B 0,C 180,E1 28362.697,E2 28362.697} C_VEL
LIN {X 0,Y 600.186,Z 1137.907,A -85,B 0,C 180,E1 28360.462,E2 28360.462} C_VEL
LIN {X 0,Y 600.03,Z 1143.491,A -85,B 0,C 180,E1 28358.529,E2 28358.529} C_VEL
LIN {X 0,Y 599.949,Z 1148.695,A -85,B 0,C 180,E1 28356.219,E2 28356.219} C_VEL
LIN {X 0,Y 599.919,Z 1152.009,A -85,B 0,C 180,E1 28354.014,E2 28354.014} C_VEL
LIN {X 0,Y 599.907,Z 1153.903,A -85,B 0,C 180,E1 28351.91,E2 28351.91} C_VEL
LIN {X 0,Y 599.885,Z 1154.394,A -85,B 0,C 180,E1 28349.522,E2 28349.522} C_VEL
LIN {X 0,Y 599.898,Z 1153.495,A -85,B 0,C 180,E1 28347.516,E2 28347.516} C_VEL
LIN {X 0,Y 599.914,Z 1151.085,A -85,B 0,C 180,E1 28345.22,E2 28345.22} C_VEL
LIN {X 0,Y 599.972,Z 1147.102,A -85,B 0,C 180,E1 28343.012,E2 28343.012} C_VEL
LIN {X 0,Y 600.048,Z 1142.219,A -85,B 0,C 180,E1 28340.988,E2 28340.988} C_VEL
LIN {X 0,Y 600.282,Z 1134.659,A -85,B 0,C 180,E1 28338.567,E2 28338.567} C_VEL
LIN {X 0,Y 600.618,Z 1127.152,A -85,B 0,C 180,E1 28336.62,E2 28336.62} C_VEL
LIN {X 0,Y 601.173,Z 1117.42,A -85,B 0,C 180,E1 28334.468,E2 28334.468} C_VEL
LIN {X 0,Y 601.949,Z 1105.684,A -85,B 0,C 180,E1 28332.303,E2 28332.303} C_VEL
LIN {X 0,Y 602.964,Z 1092.791,A -85,B 0,C 180,E1 28330.227,E2 28330.227} C_VEL
LIN {X 0,Y 604.2,Z 1078.362,A -85,B 0,C 180,E1 28328.241,E2 28328.241} C_VEL
LIN {X 0,Y 605.637,Z 1062.969,A -85,B 0,C 180,E1 28326.39,E2 28326.39} C_VEL
LIN {X 0,Y 607.318,Z 1045.365,A -85,B 0,C 180,E1 28324.551,E2 28324.551} C_VEL
LIN {X 0,Y 609.006,Z 1028.611,A -85,B 0,C 180,E1 28323.001,E2 28323.001} C_VEL
LIN {X 0,Y 611.063,Z 1008.155,A -85,B 0,C 180,E1 28321.351,E2 28321.351} C_VEL
LIN {X 0,Y 612.884,Z 989.74,A -85,B 0,C 180,E1 28320.051,E2 28320.051} C_VEL
LIN {X 0,Y 615.106,Z 966.841,A -85,B 0,C 180,E1 28318.656,E2 28318.656} C_VEL
LIN {X 0,Y 616.815,Z 947.791,A -85,B 0,C 180,E1 28317.659,E2 28317.659} C_VEL
LIN {X 0,Y 618.689,Z 925.77,A -85,B 0,C 180,E1 28316.668,E2 28316.668} C_VEL
LIN {X 0,Y 620.314,Z 902.789,A -85,B 0,C 180,E1 28315.823,E2 28315.823} C_VEL
LIN {X 0,Y 621.836,Z 879.461,A -85,B 0,C 180,E1 28315.125,E2 28315.125} C_VEL
LIN {X 0,Y 623.057,Z 855.518,A -85,B 0,C 180,E1 28314.592,E2 28314.592} C_VEL
LIN {X 0,Y 623.829,Z 833.302,A -85,B 0,C 180,E1 28314.228,E2 28314.228} C_VEL
LIN {X 0,Y 627.913,Z 596.848,A -85,B 0,C 180,E1 28311.186,E2 28311.186} C_VEL
LIN {X 0,Y 629.761,Z 488.055,A -85,B 0,C 180,E1 28309.765,E2 28309.765} C_VEL
LIN {X 0,Y 625.255,Z 468.954,A -85,B 0,C 180,E1 28309.149,E2 28309.149} C_VEL
LIN {X 0,Y 613.689,Z 449.081,A -85,B 0,C 180,E1 28307.915,E2 28307.915} C_VEL
LIN {X 0,Y 606.429,Z 430.757,A -85,B 0,C 180,E1 28305.692,E2 28305.692} C_VEL
LIN {X 0,Y 601.132,Z 417.539,A -85,B 0,C 180,E1 28303.949,E2 28303.949} C_VEL
LIN {X 0,Y 601.131,Z 417.281,A -85,B 0,C 180,E1 28300.947,E2 28300.947} C_VEL
LIN {X 0,Y 601.119,Z 417.347,A -85,B 0,C 180,E1 28297.744,E2 28297.744} C_VEL
LIN {X 0,Y 601.112,Z 417.354,A -85,B 0,C 180,E1 28294.406,E2 28294.406} C_VEL
LIN {X 0,Y 601.132,Z 417.354,A -85,B 0,C 180,E1 28291.244,E2 28291.244} C_VEL
LIN {X 0,Y 601.11,Z 417.334,A -85,B 0,C 180,E1 28288.083,E2 28288.083} C_VEL
LIN {X 0,Y 601.126,Z 417.333,A -85,B 0,C 180,E1 28284.887,E2 28284.887} C_VEL
LIN {X 0,Y 601.124,Z 417.352,A -85,B 0,C 180,E1 28281.671,E2 28281.671} C_VEL
LIN {X 0,Y 601.132,Z 417.335,A -85,B 0,C 180,E1 28278.423,E2 28278.423} C_VEL
LIN {X 0,Y 601.123,Z 417.336,A -85,B 0,C 180,E1 28275.138,E2 28275.138} C_VEL
LIN {X 0,Y 601.127,Z 417.347,A -85,B 0,C 180,E1 28271.903,E2 28271.903} C_VEL
LIN {X 0,Y 601.11,Z 417.328,A -85,B 0,C 180,E1 28268.706,E2 28268.706} C_VEL
LIN {X 0,Y 601.13,Z 417.353,A -85,B 0,C 180,E1 28265.536,E2 28265.536} C_VEL
LIN {X 0,Y 601.117,Z 417.336,A -85,B 0,C 180,E1 28262.288,E2 28262.288} C_VEL
LIN {X 0,Y 601.113,Z 417.341,A -85,B 0,C 180,E1 28258.952,E2 28258.952} C_VEL
LIN {X 0,Y 601.134,Z 417.341,A -85,B 0,C 180,E1 28255.707,E2 28255.707} C_VEL
LIN {X 0,Y 601.094,Z 417.332,A -85,B 0,C 180,E1 28252.545,E2 28252.545} C_VEL
LIN {X 0,Y 601.136,Z 417.35,A -85,B 0,C 180,E1 28249.36,E2 28249.36} C_VEL
LIN {X 0,Y 601.087,Z 417.33,A -85,B 0,C 180,E1 28246.239,E2 28246.239} C_VEL
LIN {X 0,Y 601.123,Z 417.349,A -85,B 0,C 180,E1 28243.027,E2 28243.027} C_VEL
LIN {X 0,Y 601.092,Z 417.342,A -85,B 0,C 180,E1 28239.96,E2 28239.96} C_VEL
LIN {X 0,Y 601.089,Z 417.333,A -85,B 0,C 180,E1 28236.67,E2 28236.67} C_VEL
LIN {X 0,Y 601.097,Z 417.352,A -85,B 0,C 180,E1 28233.715,E2 28233.715} C_VEL
LIN {X 0,Y 601.076,Z 417.348,A -85,B 0,C 180,E1 28230.46,E2 28230.46} C_VEL
LIN {X 0,Y 601.089,Z 417.343,A -85,B 0,C 180,E1 28227.613,E2 28227.613} C_VEL
LIN {X 0,Y 601.068,Z 417.353,A -85,B 0,C 180,E1 28224.392,E2 28224.392} C_VEL
LIN {X 0,Y 601.09,Z 417.356,A -85,B 0,C 180,E1 28221.429,E2 28221.429} C_VEL
LIN {X 0,Y 601.05,Z 417.292,A -85,B 0,C 180,E1 28218.284,E2 28218.284} C_VEL
LIN {X 0,Y 601.074,Z 417.353,A -85,B 0,C 180,E1 28215.397,E2 28215.397} C_VEL
LIN {X 0,Y 601.042,Z 417.296,A -85,B 0,C 180,E1 28212.229,E2 28212.229} C_VEL
LIN {X 0,Y 601.075,Z 417.584,A -85,B 0,C 180,E1 28210.168,E2 28210.168} C_VEL
LIN {X 0,Y 601.387,Z 418.887,A -85,B 0,C 180,E1 28210.017,E2 28210.017} C_VEL
LIN {X 0,Y 603.402,Z 422.107,A -85,B 0,C 180,E1 28209.782,E2 28209.782} C_VEL
LIN {X 0,Y 604.826,Z 424.139,A -85,B 0,C 180,E1 28209.63,E2 28209.63} C_VEL
LIN {X 0,Y 612.548,Z 435.594,A -85,B 0,C 180,E1 28208.81,E2 28208.81} C_VEL
LIN {X 0,Y 628.954,Z 462.115,A -85,B 0,C 180,E1 28207.13,E2 28207.13} C_VEL
LIN {X 0,Y 630.084,Z 464.549,A -85,B 0,C 180,E1 28207.009,E2 28207.009} C_VEL
LIN {X 0,Y 629.215,Z 510.082,A -85,B 0,C 180,E1 28206.416,E2 28206.416} C_VEL
LIN {X 0,Y 628.288,Z 517.778,A -85,B 0,C 180,E1 28206.373,E2 28206.373} C_VEL
LIN {X 0,Y 623.043,Z 538.342,A -85,B 0,C 180,E1 28206.465,E2 28206.465} C_VEL
LIN {X 0,Y 622.311,Z 544.948,A -85,B 0,C 180,E1 28206.423,E2 28206.423} C_VEL
LIN {X 0,Y 617.501,Z 798.266,A -85,B 0,C 180,E1 28203.131,E2 28203.131} C_VEL
LIN {X 0,Y 616.712,Z 820.342,A -85,B 0,C 180,E1 28202.76,E2 28202.76} C_VEL
LIN {X 0,Y 615.428,Z 845.487,A -85,B 0,C 180,E1 28202.172,E2 28202.172} C_VEL
LIN {X 0,Y 614.03,Z 866.815,A -85,B 0,C 180,E1 28201.515,E2 28201.515} C_VEL
LIN {X 0,Y 612.369,Z 889.06,A -85,B 0,C 180,E1 28200.681,E2 28200.681} C_VEL
LIN {X 0,Y 610.434,Z 910.412,A -85,B 0,C 180,E1 28199.703,E2 28199.703} C_VEL
LIN {X 0,Y 608.564,Z 929.738,A -85,B 0,C 180,E1 28198.67,E2 28198.67} C_VEL
LIN {X 0,Y 606.223,Z 951.833,A -85,B 0,C 180,E1 28197.292,E2 28197.292} C_VEL
LIN {X 0,Y 604.204,Z 970.239,A -85,B 0,C 180,E1 28195.959,E2 28195.959} C_VEL
LIN {X 0,Y 601.852,Z 990.992,A -85,B 0,C 180,E1 28194.227,E2 28194.227} C_VEL
